LIN {X 0,Y 163.104,Z 333.396,A -85,B 0,C 180,E1 -26252.044,E2 -26252.044} C_VEL
LIN {X 0,Y 169.371,Z 321.967,A -85,B 0,C 180,E1 -26253.809,E2 -26253.809} C_VEL
LIN {X 0,Y 174.292,Z 311.209,A -85,B 0,C 180,E1 -26255.131,E2 -26255.131} C_VEL
LIN {X 0,Y 179.303,Z 297.656,A -85,B 0,C 180,E1 -26256.379,E2 -26256.379} C_VEL
LIN {X 0,Y 183.251,Z 283.24,A -85,B 0,C 180,E1 -26257.382,E2 -26257.382} C_VEL
LIN {X 0,Y 185.938,Z 269.575,A -85,B 0,C 180,E1 -26257.977,E2 -26257.977} C_VEL
LIN {X 0,Y 188.353,Z 247.435,A -85,B 0,C 180,E1 -26258.617,E2 -26258.617} C_VEL
LIN {X 0,Y 189.054,Z 239.838,A -85,B 0,C 180,E1 -26258.835,E2 -26258.835} C_VEL
LIN {X 0,Y 185.822,Z 232.857,A -85,B 0,C 180,E1 -26261.889,E2 -26261.889} C_VEL
LIN {X 0,Y 182.763,Z 226.917,A -85,B 0,C 180,E1 -26265.276,E2 -26265.276} C_VEL
LIN {X 0,Y 180.995,Z 223.675,A -85,B 0,C 180,E1 -26267.597,E2 -26267.597} C_VEL
LIN {X 0,Y 179.349,Z 220.559,A -85,B 0,C 180,E1 -26270.198,E2 -26270.198} C_VEL
LIN {X 0,Y 177.583,Z 217.018,A -85,B 0,C 180,E1 -26273.894,E2 -26273.894} C_VEL
LIN {X 0,Y 175.962,Z 213.489,A -85,B 0,C 180,E1 -26280.646,E2 -26280.646} C_VEL
LIN {X 0,Y 175.948,Z 212.764,A -85,B 0,C 180,E1 -26281.791,E2 -26281.791} C_VEL
LIN {X 0,Y 175.948,Z 213.169,A -85,B 0,C 180,E1 -26284.582,E2 -26284.582} C_VEL
LIN {X 0,Y 177.027,Z 216.627,A -85,B 0,C 180,E1 -26290.503,E2 -26290.503} C_VEL
LIN {X 0,Y 177.831,Z 217.67,A -85,B 0,C 180,E1 -26292.481,E2 -26292.481} C_VEL
LIN {X 0,Y 180.086,Z 221.968,A -85,B 0,C 180,E1 -26296.763,E2 -26296.763} C_VEL
LIN {X 0,Y 182.173,Z 225.802,A -85,B 0,C 180,E1 -26299.713,E2 -26299.713} C_VEL
LIN {X 0,Y 183.869,Z 229.479,A -85,B 0,C 180,E1 -26301.807,E2 -26301.807} C_VEL
LIN {X 0,Y 186.407,Z 236.279,A -85,B 0,C 180,E1 -26304.65,E2 -26304.65} C_VEL
LIN {X 0,Y 188.76,Z 243.058,A -85,B 0,C 180,E1 -26306.989,E2 -26306.989} C_VEL
LIN {X 0,Y 185.981,Z 270.935,A -85,B 0,C 180,E1 -26307.786,E2 -26307.786} C_VEL
LIN {X 0,Y 183.211,Z 285.581,A -85,B 0,C 180,E1 -26308.371,E2 -26308.371} C_VEL
LIN {X 0,Y 179.573,Z 298.889,A -85,B 0,C 180,E1 -26309.161,E2 -26309.161} C_VEL
LIN {X 0,Y 174.882,Z 311.931,A -85,B 0,C 180,E1 -26310.228,E2 -26310.228} C_VEL
LIN {X 0,Y 169.208,Z 324.559,A -85,B 0,C 180,E1 -26311.628,E2 -26311.628} C_VEL
LIN {X 0,Y 162.997,Z 336.072,A -85,B 0,C 180,E1 -26313.342,E2 -26313.342} C_VEL
LIN {X 0,Y 155.623,Z 347.616,A -85,B 0,C 180,E1 -26315.621,E2 -26315.621} C_VEL
LIN {X 0,Y 147.797,Z 358.182,A -85,B 0,C 180,E1 -26318.474,E2 -26318.474} C_VEL
LIN {X 0,Y 140.729,Z 366.499,A -85,B 0,C 180,E1 -26321.487,E2 -26321.487} C_VEL
LIN {X 0,Y 132.765,Z 374.701,A -85,B 0,C 180,E1 -26325.46,E2 -26325.46} C_VEL
LIN {X 0,Y 125.61,Z 381.317,A -85,B 0,C 180,E1 -26329.951,E2 -26329.951} C_VEL
LIN {X 0,Y 118.469,Z 387.209,A -85,B 0,C 180,E1 -26335.696,E2 -26335.696} C_VEL
LIN {X 0,Y 114.158,Z 390.634,A -85,B 0,C 180,E1 -26340.494,E2 -26340.494} C_VEL
LIN {X 0,Y 109.512,Z 393.899,A -85,B 0,C 180,E1 -26347.352,E2 -26347.352} C_VEL
LIN {X 0,Y 106.522,Z 395.797,A -85,B 0,C 180,E1 -26354.697,E2 -26354.697} C_VEL
LIN {X 0,Y 105.175,Z 396.381,A -85,B 0,C 180,E1 -26362.319,E2 -26362.319} C_VEL
LIN {X 0,Y 105.031,Z 396.178,A -85,B 0,C 180,E1 -26366.163,E2 -26366.163} C_VEL
LIN {X 0,Y 105.107,Z 395.641,A -85,B 0,C 180,E1 -26369.999,E2 -26369.999} C_VEL
LIN {X 0,Y 105.019,Z 394.753,A -85,B 0,C 180,E1 -26373.837,E2 -26373.837} C_VEL
LIN {X 0,Y 105.593,Z 391.925,A -85,B 0,C 180,E1 -26381.517,E2 -26381.517} C_VEL
LIN {X 0,Y 107.551,Z 387.625,A -85,B 0,C 180,E1 -26389.07,E2 -26389.07} C_VEL
LIN {X 0,Y 110.164,Z 383.371,A -85,B 0,C 180,E1 -26394.498,E2 -26394.498} C_VEL
LIN {X 0,Y 112.428,Z 379.759,A -85,B 0,C 180,E1 -26398.193,E2 -26398.193} C_VEL
LIN {X 0,Y 113.595,Z 377.02,A -85,B 0,C 180,E1 -26400.781,E2 -26400.781} C_VEL
LIN {X 0,Y 114.307,Z 372.208,A -85,B 0,C 180,E1 -26405.14,E2 -26405.14} C_VEL
LIN {X 0,Y 115.529,Z 366.929,A -85,B 0,C 180,E1 -26409.276,E2 -26409.276} C_VEL
LIN {X 0,Y 117.403,Z 363.367,A -85,B 0,C 180,E1 -26411.41,E2 -26411.41} C_VEL
LIN {X 0,Y 123.341,Z 354.399,A -85,B 0,C 180,E1 -26415.418,E2 -26415.418} C_VEL
LIN {X 0,Y 129.458,Z 344.175,A -85,B 0,C 180,E1 -26418.871,E2 -26418.871} C_VEL
LIN {X 0,Y 135.274,Z 332.907,A -85,B 0,C 180,E1 -26421.794,E2 -26421.794} C_VEL
LIN {X 0,Y 140.868,Z 320.442,A -85,B 0,C 180,E1 -26424.166,E2 -26424.166} C_VEL
LIN {X 0,Y 145.747,Z 307.43,A -85,B 0,C 180,E1 -26425.974,E2 -26425.974} C_VEL
LIN {X 0,Y 149.74,Z 293.962,A -85,B 0,C 180,E1 -26427.339,E2 -26427.339} C_VEL
LIN {X 0,Y 152.837,Z 279.632,A -85,B 0,C 180,E1 -26428.369,E2 -26428.369} C_VEL
LIN {X 0,Y 154.871,Z 265.326,A -85,B 0,C 180,E1 -26428.993,E2 -26428.993} C_VEL
LIN {X 0,Y 158.466,Z 223.489,A -85,B 0,C 180,E1 -26430.437,E2 -26430.437} C_VEL
LIN {X 0,Y 154.926,Z 212.982,A -85,B 0,C 180,E1 -26433.497,E2 -26433.497} C_VEL
LIN {X 0,Y 152.921,Z 208.654,A -85,B 0,C 180,E1 -26435.273,E2 -26435.273} C_VEL
LIN {X 0,Y 149.061,Z 201.739,A -85,B 0,C 180,E1 -26439.021,E2 -26439.021} C_VEL
LIN {X 0,Y 145.805,Z 196.184,A -85,B 0,C 180,E1 -26442.829,E2 -26442.829} C_VEL
LIN {X 0,Y 143.005,Z 191.844,A -85,B 0,C 180,E1 -26446.863,E2 -26446.863} C_VEL
LIN {X 0,Y 140.93,Z 188.345,A -85,B 0,C 180,E1 -26450.854,E2 -26450.854} C_VEL
LIN {X 0,Y 140.403,Z 187.555,A -85,B 0,C 180,E1 -26452.088,E2 -26452.088} C_VEL
LIN {X 0,Y 138.478,Z 184.233,A -85,B 0,C 180,E1 -26459.546,E2 -26459.546} C_VEL
LIN {X 0,Y 138.413,Z 182.933,A -85,B 0,C 180,E1 -26461.609,E2 -26461.609} C_VEL
LIN {X 0,Y 138.346,Z 183.294,A -85,B 0,C 180,E1 -26464.371,E2 -26464.371} C_VEL
LIN {X 0,Y 139.797,Z 187.241,A -85,B 0,C 180,E1 -26472.837,E2 -26472.837} C_VEL
LIN {X 0,Y 140.818,Z 188.256,A -85,B 0,C 180,E1 -26475.286,E2 -26475.286} C_VEL
LIN {X 0,Y 142.811,Z 191.691,A -85,B 0,C 180,E1 -26479.215,E2 -26479.215} C_VEL
LIN {X 0,Y 143.828,Z 193.178,A -85,B 0,C 180,E1 -26480.816,E2 -26480.816} C_VEL
LIN {X 0,Y 146.549,Z 197.585,A -85,B 0,C 180,E1 -26484.506,E2 -26484.506} C_VEL
LIN {X 0,Y 149.425,Z 202.393,A -85,B 0,C 180,E1 -26487.739,E2 -26487.739} C_VEL
LIN {X 0,Y 153.193,Z 209.339,A -85,B 0,C 180,E1 -26491.362,E2 -26491.362} C_VEL
LIN {X 0,Y 157.413,Z 217.975,A -85,B 0,C 180,E1 -26494.866,E2 -26494.866} C_VEL
LIN {X 0,Y 158.652,Z 220.72,A -85,B 0,C 180,E1 -26495.815,E2 -26495.815} C_VEL
LIN {X 0,Y 154.442,Z 267.31,A -85,B 0,C 180,E1 -26497.421,E2 -26497.421} C_VEL
LIN {X 0,Y 152.166,Z 281.337,A -85,B 0,C 180,E1 -26498.264,E2 -26498.264} C_VEL
LIN {X 0,Y 148.978,Z 294.723,A -85,B 0,C 180,E1 -26499.423,E2 -26499.423} C_VEL
LIN {X 0,Y 144.539,Z 308.698,A -85,B 0,C 180,E1 -26501.092,E2 -26501.092} C_VEL
LIN {X 0,Y 139.567,Z 321.183,A -85,B 0,C 180,E1 -26503.101,E2 -26503.101} C_VEL
LIN {X 0,Y 134.272,Z 332.561,A -85,B 0,C 180,E1 -26505.568,E2 -26505.568} C_VEL
LIN {X 0,Y 128.123,Z 343.987,A -85,B 0,C 180,E1 -26508.835,E2 -26508.835} C_VEL
LIN {X 0,Y 121.827,Z 354.21,A -85,B 0,C 180,E1 -26512.719,E2 -26512.719} C_VEL
LIN {X 0,Y 116.131,Z 362.66,A -85,B 0,C 180,E1 -26516.999,E2 -26516.999} C_VEL
LIN {X 0,Y 110.441,Z 370.728,A -85,B 0,C 180,E1 -26522.526,E2 -26522.526} C_VEL
LIN {X 0,Y 105.679,Z 377.239,A -85,B 0,C 180,E1 -26528.546,E2 -26528.546} C_VEL
LIN {X 0,Y 102.369,Z 381.755,A -85,B 0,C 180,E1 -26534.062,E2 -26534.062} C_VEL
LIN {X 0,Y 99.52,Z 386.369,A -85,B 0,C 180,E1 -26541.881,E2 -26541.881} C_VEL
LIN {X 0,Y 98.141,Z 389.507,A -85,B 0,C 180,E1 -26550.001,E2 -26550.001} C_VEL
LIN {X 0,Y 97.843,Z 390.569,A -85,B 0,C 180,E1 -26554.12,E2 -26554.12} C_VEL
LIN {X 0,Y 98.05,Z 391.703,A -85,B 0,C 180,E1 -26562.418,E2 -26562.418} C_VEL
LIN {X 0,Y 99.812,Z 391.512,A -85,B 0,C 180,E1 -26570.614,E2 -26570.614} C_VEL
LIN {X 0,Y 103.186,Z 389.978,A -85,B 0,C 180,E1 -26578.475,E2 -26578.475} C_VEL
LIN {X 0,Y 108.115,Z 387.062,A -85,B 0,C 180,E1 -26585.807,E2 -26585.807} C_VEL
LIN {X 0,Y 114.599,Z 382.674,A -85,B 0,C 180,E1 -26592.424,E2 -26592.424} C_VEL
LIN {X 0,Y 120.346,Z 378.294,A -85,B 0,C 180,E1 -26596.885,E2 -26596.885} C_VEL
LIN {X 0,Y 127.866,Z 371.916,A -85,B 0,C 180,E1 -26601.558,E2 -26601.558} C_VEL
LIN {X 0,Y 134.906,Z 365.106,A -85,B 0,C 180,E1 -26605.229,E2 -26605.229} C_VEL
LIN {X 0,Y 142.286,Z 357.096,A -85,B 0,C 180,E1 -26608.434,E2 -26608.434} C_VEL
LIN {X 0,Y 150.264,Z 347.31,A -85,B 0,C 180,E1 -26611.278,E2 -26611.278} C_VEL
LIN {X 0,Y 157.794,Z 336.411,A -85,B 0,C 180,E1 -26613.683,E2 -26613.683} C_VEL
LIN {X 0,Y 164.151,Z 325.597,A -85,B 0,C 180,E1 -26615.479,E2 -26615.479} C_VEL
LIN {X 0,Y 169.948,Z 313.913,A -85,B 0,C 180,E1 -26616.944,E2 -26616.944} C_VEL
LIN {X 0,Y 175.446,Z 300.22,A -85,B 0,C 180,E1 -26618.233,E2 -26618.233} C_VEL
LIN {X 0,Y 179.521,Z 286.575,A -85,B 0,C 180,E1 -26619.238,E2 -26619.238} C_VEL
LIN {X 0,Y 182.66,Z 272.102,A -85,B 0,C 180,E1 -26619.899,E2 -26619.899} C_VEL
LIN {X 0,Y 184.777,Z 255.073,A -85,B 0,C 180,E1 -26620.423,E2 -26620.423} C_VEL
LIN {X 0,Y 185.896,Z 243.533,A -85,B 0,C 180,E1 -26620.735,E2 -26620.735} C_VEL
LIN {X 0,Y 182.864,Z 236.776,A -85,B 0,C 180,E1 -26623.973,E2 -26623.973} C_VEL
LIN {X 0,Y 180.035,Z 231.055,A -85,B 0,C 180,E1 -26627.619,E2 -26627.619} C_VEL
LIN {X 0,Y 178.151,Z 227.388,A -85,B 0,C 180,E1 -26630.688,E2 -26630.688} C_VEL
LIN {X 0,Y 176.418,Z 223.824,A -85,B 0,C 180,E1 -26634.57,E2 -26634.57} C_VEL
LIN {X 0,Y 175.062,Z 220.259,A -85,B 0,C 180,E1 -26641.3,E2 -26641.3} C_VEL
LIN {X 0,Y 175.065,Z 219.76,A -85,B 0,C 180,E1 -26642.3,E2 -26642.3} C_VEL
LIN {X 0,Y 175.059,Z 220.213,A -85,B 0,C 180,E1 -26644.317,E2 -26644.317} C_VEL
LIN {X 0,Y 176.046,Z 223.603,A -85,B 0,C 180,E1 -26650.218,E2 -26650.218} C_VEL
LIN {X 0,Y 176.695,Z 224.506,A -85,B 0,C 180,E1 -26651.925,E2 -26651.925} C_VEL
LIN {X 0,Y 178.723,Z 228.592,A -85,B 0,C 180,E1 -26656.069,E2 -26656.069} C_VEL
LIN {X 0,Y 180.56,Z 232.171,A -85,B 0,C 180,E1 -26658.866,E2 -26658.866} C_VEL
LIN {X 0,Y 181.999,Z 235.567,A -85,B 0,C 180,E1 -26660.798,E2 -26660.798} C_VEL
LIN {X 0,Y 184.301,Z 242.191,A -85,B 0,C 180,E1 -26663.604,E2 -26663.604} C_VEL
LIN {X 0,Y 185.669,Z 246.321,A -85,B 0,C 180,E1 -26665.101,E2 -26665.101} C_VEL
LIN {X 0,Y 182.99,Z 271.487,A -85,B 0,C 180,E1 -26665.793,E2 -26665.793} C_VEL
LIN {X 0,Y 180.159,Z 285.904,A -85,B 0,C 180,E1 -26666.361,E2 -26666.361} C_VEL
LIN {X 0,Y 176.237,Z 299.649,A -85,B 0,C 180,E1 -26667.154,E2 -26667.154} C_VEL
LIN {X 0,Y 171.429,Z 312.489,A -85,B 0,C 180,E1 -26668.184,E2 -26668.184} C_VEL
LIN {X 0,Y 165.611,Z 324.977,A -85,B 0,C 180,E1 -26669.546,E2 -26669.546} C_VEL
LIN {X 0,Y 159.214,Z 336.387,A -85,B 0,C 180,E1 -26671.212,E2 -26671.212} C_VEL
LIN {X 0,Y 151.607,Z 347.848,A -85,B 0,C 180,E1 -26673.444,E2 -26673.444} C_VEL
LIN {X 0,Y 144.102,Z 357.592,A -85,B 0,C 180,E1 -26676.03,E2 -26676.03} C_VEL
LIN {X 0,Y 136.131,Z 366.605,A -85,B 0,C 180,E1 -26679.249,E2 -26679.249} C_VEL
LIN {X 0,Y 127.786,Z 374.742,A -85,B 0,C 180,E1 -26683.22,E2 -26683.22} C_VEL
LIN {X 0,Y 120.231,Z 381.317,A -85,B 0,C 180,E1 -26687.76,E2 -26687.76} C_VEL
LIN {X 0,Y 112.647,Z 387.172,A -85,B 0,C 180,E1 -26693.65,E2 -26693.65} C_VEL
LIN {X 0,Y 107.974,Z 390.572,A -85,B 0,C 180,E1 -26698.619,E2 -26698.619} C_VEL
LIN {X 0,Y 102.955,Z 393.793,A -85,B 0,C 180,E1 -26705.821,E2 -26705.821} C_VEL
LIN {X 0,Y 99.658,Z 395.658,A -85,B 0,C 180,E1 -26713.615,E2 -26713.615} C_VEL
LIN {X 0,Y 98.115,Z 396.209,A -85,B 0,C 180,E1 -26721.763,E2 -26721.763} C_VEL
LIN {X 0,Y 97.935,Z 395.991,A -85,B 0,C 180,E1 -26725.884,E2 -26725.884} C_VEL
LIN {X 0,Y 98.005,Z 395.438,A -85,B 0,C 180,E1 -26729.999,E2 -26729.999} C_VEL
LIN {X 0,Y 97.925,Z 394.533,A -85,B 0,C 180,E1 -26734.115,E2 -26734.115} C_VEL
LIN {X 0,Y 98.62,Z 391.671,A -85,B 0,C 180,E1 -26742.344,E2 -26742.344} C_VEL
LIN {X 0,Y 100.822,Z 387.334,A -85,B 0,C 180,E1 -26750.397,E2 -26750.397} C_VEL
LIN {X 0,Y 103.673,Z 383.041,A -85,B 0,C 180,E1 -26756.144,E2 -26756.144} C_VEL
LIN {X 0,Y 107.997,Z 376.757,A -85,B 0,C 180,E1 -26762.471,E2 -26762.471} C_VEL
LIN {X 0,Y 113.59,Z 368.924,A -85,B 0,C 180,E1 -26768.222,E2 -26768.222} C_VEL
LIN {X 0,Y 117.403,Z 363.367,A -85,B 0,C 180,E1 -26771.41,E2 -26771.41} C_VEL
LIN {X 0,Y 119.402,Z 359.663,A -85,B 0,C 180,E1 -26773.418,E2 -26773.418} C_VEL
LIN {X 0,Y 121.462,Z 353.381,A -85,B 0,C 180,E1 -26776.931,E2 -26776.931} C_VEL
LIN {X 0,Y 123.614,Z 346.643,A -85,B 0,C 180,E1 -26780.18,E2 -26780.18} C_VEL
LIN {X 0,Y 125.657,Z 342.225,A -85,B 0,C 180,E1 -26781.723,E2 -26781.723} C_VEL
LIN {X 0,Y 131.589,Z 330.916,A -85,B 0,C 180,E1 -26784.535,E2 -26784.535} C_VEL
LIN {X 0,Y 137.479,Z 318.039,A -85,B 0,C 180,E1 -26786.834,E2 -26786.834} C_VEL
LIN {X 0,Y 142.217,Z 305.453,A -85,B 0,C 180,E1 -26788.478,E2 -26788.478} C_VEL
LIN {X 0,Y 146.366,Z 291.429,A -85,B 0,C 180,E1 -26789.802,E2 -26789.802} C_VEL
LIN {X 0,Y 149.297,Z 277.579,A -85,B 0,C 180,E1 -26790.723,E2 -26790.723} C_VEL
LIN {X 0,Y 151.247,Z 263,A -85,B 0,C 180,E1 -26791.307,E2 -26791.307} C_VEL
LIN {X 0,Y 154.515,Z 225.964,A -85,B 0,C 180,E1 -26792.58,E2 -26792.58} C_VEL
LIN {X 0,Y 151.565,Z 216.879,A -85,B 0,C 180,E1 -26795.426,E2 -26795.426} C_VEL
LIN {X 0,Y 148.637,Z 210.986,A -85,B 0,C 180,E1 -26798.322,E2 -26798.322} C_VEL
LIN {X 0,Y 145.667,Z 205.538,A -85,B 0,C 180,E1 -26801.701,E2 -26801.701} C_VEL
LIN {X 0,Y 143.432,Z 201.744,A -85,B 0,C 180,E1 -26804.685,E2 -26804.685} C_VEL
LIN {X 0,Y 141.599,Z 198.533,A -85,B 0,C 180,E1 -26807.641,E2 -26807.641} C_VEL
LIN {X 0,Y 139.596,Z 194.873,A -85,B 0,C 180,E1 -26811.86,E2 -26811.86} C_VEL
LIN {X 0,Y 137.523,Z 190.884,A -85,B 0,C 180,E1 -26820.592,E2 -26820.592} C_VEL
LIN {X 0,Y 137.523,Z 189.96,A -85,B 0,C 180,E1 -26822.056,E2 -26822.056} C_VEL
LIN {X 0,Y 137.465,Z 190.509,A -85,B 0,C 180,E1 -26824.491,E2 -26824.491} C_VEL
LIN {X 0,Y 138.714,Z 194.154,A -85,B 0,C 180,E1 -26832.283,E2 -26832.283} C_VEL
LIN {X 0,Y 139.651,Z 195.224,A -85,B 0,C 180,E1 -26834.715,E2 -26834.715} C_VEL
LIN {X 0,Y 141.692,Z 198.729,A -85,B 0,C 180,E1 -26838.903,E2 -26838.903} C_VEL
LIN {X 0,Y 144.63,Z 203.761,A -85,B 0,C 180,E1 -26843.351,E2 -26843.351} C_VEL
LIN {X 0,Y 147.643,Z 209.116,A -85,B 0,C 180,E1 -26846.983,E2 -26846.983} C_VEL
LIN {X 0,Y 151.266,Z 216.339,A -85,B 0,C 180,E1 -26850.678,E2 -26850.678} C_VEL
LIN {X 0,Y 154.668,Z 223.78,A -85,B 0,C 180,E1 -26853.696,E2 -26853.696} C_VEL
LIN {X 0,Y 150.612,Z 267.23,A -85,B 0,C 180,E1 -26855.186,E2 -26855.186} C_VEL
LIN {X 0,Y 148.219,Z 281.466,A -85,B 0,C 180,E1 -26856.024,E2 -26856.024} C_VEL
LIN {X 0,Y 144.94,Z 294.764,A -85,B 0,C 180,E1 -26857.153,E2 -26857.153} C_VEL
LIN {X 0,Y 140.67,Z 307.884,A -85,B 0,C 180,E1 -26858.682,E2 -26858.682} C_VEL
LIN {X 0,Y 135.483,Z 320.559,A -85,B 0,C 180,E1 -26860.655,E2 -26860.655} C_VEL
LIN {X 0,Y 129.928,Z 332.078,A -85,B 0,C 180,E1 -26863.095,E2 -26863.095} C_VEL
LIN {X 0,Y 124.04,Z 342.643,A -85,B 0,C 180,E1 -26866.047,E2 -26866.047} C_VEL
LIN {X 0,Y 117.336,Z 353.131,A -85,B 0,C 180,E1 -26869.919,E2 -26869.919} C_VEL
LIN {X 0,Y 111.209,Z 361.787,A -85,B 0,C 180,E1 -26874.229,E2 -26874.229} C_VEL
LIN {X 0,Y 105.012,Z 370.089,A -85,B 0,C 180,E1 -26879.872,E2 -26879.872} C_VEL
LIN {X 0,Y 100.448,Z 375.875,A -85,B 0,C 180,E1 -26885.179,E2 -26885.179} C_VEL
LIN {X 0,Y 95.592,Z 382.074,A -85,B 0,C 180,E1 -26892.898,E2 -26892.898} C_VEL
LIN {X 0,Y 92.508,Z 386.632,A -85,B 0,C 180,E1 -26901.261,E2 -26901.261} C_VEL
LIN {X 0,Y 91.04,Z 389.732,A -85,B 0,C 180,E1 -26910.001,E2 -26910.001} C_VEL
LIN {X 0,Y 90.744,Z 390.777,A -85,B 0,C 180,E1 -26914.443,E2 -26914.443} C_VEL
LIN {X 0,Y 91.052,Z 391.877,A -85,B 0,C 180,E1 -26923.39,E2 -26923.39} C_VEL
LIN {X 0,Y 93.092,Z 391.65,A -85,B 0,C 180,E1 -26932.178,E2 -26932.178} C_VEL
LIN {X 0,Y 96.881,Z 390.08,A -85,B 0,C 180,E1 -26940.518,E2 -26940.518} C_VEL
LIN {X 0,Y 102.327,Z 387.127,A -85,B 0,C 180,E1 -26948.181,E2 -26948.181} C_VEL
LIN {X 0,Y 109.457,Z 382.637,A -85,B 0,C 180,E1 -26955.065,E2 -26955.065} C_VEL
LIN {X 0,Y 115.535,Z 378.277,A -85,B 0,C 180,E1 -26959.498,E2 -26959.498} C_VEL
LIN {X 0,Y 123.506,Z 371.855,A -85,B 0,C 180,E1 -26964.183,E2 -26964.183} C_VEL
LIN {X 0,Y 132.116,Z 363.844,A -85,B 0,C 180,E1 -26968.335,E2 -26968.335} C_VEL
LIN {X 0,Y 140.02,Z 355.434,A -85,B 0,C 180,E1 -26971.448,E2 -26971.448} C_VEL
LIN {X 0,Y 148.368,Z 345.281,A -85,B 0,C 180,E1 -26974.16,E2 -26974.16} C_VEL
LIN {X 0,Y 156.156,Z 333.853,A -85,B 0,C 180,E1 -26976.492,E2 -26976.492} C_VEL
LIN {X 0,Y 162.803,Z 322.461,A -85,B 0,C 180,E1 -26978.146,E2 -26978.146} C_VEL
LIN {X 0,Y 168.757,Z 309.962,A -85,B 0,C 180,E1 -26979.559,E2 -26979.559} C_VEL
LIN {X 0,Y 173.789,Z 296.759,A -85,B 0,C 180,E1 -26980.655,E2 -26980.655} C_VEL
LIN {X 0,Y 177.656,Z 283.154,A -85,B 0,C 180,E1 -26981.525,E2 -26981.525} C_VEL
LIN {X 0,Y 180.521,Z 268.984,A -85,B 0,C 180,E1 -26982.088,E2 -26982.088} C_VEL
LIN {X 0,Y 182.949,Z 247.322,A -85,B 0,C 180,E1 -26982.689,E2 -26982.689} C_VEL
LIN {X 0,Y 179.944,Z 240.491,A -85,B 0,C 180,E1 -26986.375,E2 -26986.375} C_VEL
LIN {X 0,Y 177.768,Z 236.075,A -85,B 0,C 180,E1 -26989.673,E2 -26989.673} C_VEL
LIN {X 0,Y 176.761,Z 233.861,A -85,B 0,C 180,E1 -26991.584,E2 -26991.584} C_VEL
LIN {X 0,Y 175.333,Z 230.66,A -85,B 0,C 180,E1 -26995.113,E2 -26995.113} C_VEL
LIN {X 0,Y 174.181,Z 227.13,A -85,B 0,C 180,E1 -27001.809,E2 -27001.809} C_VEL
LIN {X 0,Y 174.196,Z 226.822,A -85,B 0,C 180,E1 -27002.312,E2 -27002.312} C_VEL
LIN {X 0,Y 174.176,Z 227.232,A -85,B 0,C 180,E1 -27004.049,E2 -27004.049} C_VEL
LIN {X 0,Y 175.071,Z 230.567,A -85,B 0,C 180,E1 -27009.93,E2 -27009.93} C_VEL
LIN {X 0,Y 175.595,Z 231.377,A -85,B 0,C 180,E1 -27011.412,E2 -27011.412} C_VEL
LIN {X 0,Y 177.469,Z 235.394,A -85,B 0,C 180,E1 -27015.517,E2 -27015.517} C_VEL
LIN {X 0,Y 179.295,Z 239.222,A -85,B 0,C 180,E1 -27018.457,E2 -27018.457} C_VEL
LIN {X 0,Y 181.083,Z 244.267,A -85,B 0,C 180,E1 -27021,E2 -27021} C_VEL
LIN {X 0,Y 182.759,Z 249.639,A -85,B 0,C 180,E1 -27023.136,E2 -27023.136} C_VEL
LIN {X 0,Y 180.234,Z 272.031,A -85,B 0,C 180,E1 -27023.74,E2 -27023.74} C_VEL
LIN {X 0,Y 177.326,Z 286.234,A -85,B 0,C 180,E1 -27024.277,E2 -27024.277} C_VEL
LIN {X 0,Y 173.128,Z 300.412,A -85,B 0,C 180,E1 -27025.074,E2 -27025.074} C_VEL
LIN {X 0,Y 168.208,Z 313.05,A -85,B 0,C 180,E1 -27026.063,E2 -27026.063} C_VEL
LIN {X 0,Y 162.244,Z 325.398,A -85,B 0,C 180,E1 -27027.375,E2 -27027.375} C_VEL
LIN {X 0,Y 154.941,Z 337.871,A -85,B 0,C 180,E1 -27029.171,E2 -27029.171} C_VEL
LIN {X 0,Y 147.813,Z 348.086,A -85,B 0,C 180,E1 -27031.147,E2 -27031.147} C_VEL
LIN {X 0,Y 140.496,Z 357.217,A -85,B 0,C 180,E1 -27033.523,E2 -27033.523} C_VEL
LIN {X 0,Y 131.746,Z 366.703,A -85,B 0,C 180,E1 -27036.853,E2 -27036.853} C_VEL
LIN {X 0,Y 123.023,Z 374.784,A -85,B 0,C 180,E1 -27040.804,E2 -27040.804} C_VEL
LIN {X 0,Y 115.049,Z 381.318,A -85,B 0,C 180,E1 -27045.372,E2 -27045.372} C_VEL
LIN {X 0,Y 106.984,Z 387.134,A -85,B 0,C 180,E1 -27051.385,E2 -27051.385} C_VEL
LIN {X 0,Y 101.923,Z 390.504,A -85,B 0,C 180,E1 -27056.52,E2 -27056.52} C_VEL
LIN {X 0,Y 96.486,Z 393.686,A -85,B 0,C 180,E1 -27064.084,E2 -27064.084} C_VEL
LIN {X 0,Y 92.842,Z 395.519,A -85,B 0,C 180,E1 -27072.374,E2 -27072.374} C_VEL
LIN {X 0,Y 91.081,Z 396.038,A -85,B 0,C 180,E1 -27081.122,E2 -27081.122} C_VEL
LIN {X 0,Y 90.862,Z 395.804,A -85,B 0,C 180,E1 -27085.563,E2 -27085.563} C_VEL
LIN {X 0,Y 90.911,Z 395.234,A -85,B 0,C 180,E1 -27089.999,E2 -27089.999} C_VEL
LIN {X 0,Y 90.825,Z 394.312,A -85,B 0,C 180,E1 -27094.437,E2 -27094.437} C_VEL
LIN {X 0,Y 91.648,Z 391.415,A -85,B 0,C 180,E1 -27103.299,E2 -27103.299} C_VEL
LIN {X 0,Y 94.162,Z 387.044,A -85,B 0,C 180,E1 -27111.911,E2 -27111.911} C_VEL
LIN {X 0,Y 97.283,Z 382.711,A -85,B 0,C 180,E1 -27118.006,E2 -27118.006} C_VEL
LIN {X 0,Y 102.017,Z 376.386,A -85,B 0,C 180,E1 -27124.634,E2 -27124.634} C_VEL
LIN {X 0,Y 108.039,Z 368.506,A -85,B 0,C 180,E1 -27130.579,E2 -27130.579} C_VEL
LIN {X 0,Y 114.002,Z 360.267,A -85,B 0,C 180,E1 -27135.149,E2 -27135.149} C_VEL
LIN {X 0,Y 120.717,Z 350.342,A -85,B 0,C 180,E1 -27139.186,E2 -27139.186} C_VEL
LIN {X 0,Y 125.657,Z 342.225,A -85,B 0,C 180,E1 -27141.723,E2 -27141.723} C_VEL
LIN {X 0,Y 127.665,Z 337.74,A -85,B 0,C 180,E1 -27143.183,E2 -27143.183} C_VEL
LIN {X 0,Y 129.727,Z 330.204,A -85,B 0,C 180,E1 -27145.9,E2 -27145.9} C_VEL
LIN {X 0,Y 131.809,Z 322.362,A -85,B 0,C 180,E1 -27148.366,E2 -27148.366} C_VEL
LIN {X 0,Y 133.702,Z 317.246,A -85,B 0,C 180,E1 -27149.39,E2 -27149.39} C_VEL
LIN {X 0,Y 138.972,Z 303.467,A -85,B 0,C 180,E1 -27151.105,E2 -27151.105} C_VEL
LIN {X 0,Y 142.898,Z 290.17,A -85,B 0,C 180,E1 -27152.284,E2 -27152.284} C_VEL
LIN {X 0,Y 145.795,Z 276.687,A -85,B 0,C 180,E1 -27153.107,E2 -27153.107} C_VEL
LIN {X 0,Y 147.709,Z 262.134,A -85,B 0,C 180,E1 -27153.681,E2 -27153.681} C_VEL
LIN {X 0,Y 150.78,Z 228.515,A -85,B 0,C 180,E1 -27154.83,E2 -27154.83} C_VEL
LIN {X 0,Y 148.591,Z 221.499,A -85,B 0,C 180,E1 -27157.194,E2 -27157.194} C_VEL
LIN {X 0,Y 145.249,Z 214.542,A -85,B 0,C 180,E1 -27160.938,E2 -27160.938} C_VEL
LIN {X 0,Y 142.313,Z 208.97,A -85,B 0,C 180,E1 -27164.905,E2 -27164.905} C_VEL
LIN {X 0,Y 140.124,Z 205.101,A -85,B 0,C 180,E1 -27168.61,E2 -27168.61} C_VEL
LIN {X 0,Y 138.163,Z 201.308,A -85,B 0,C 180,E1 -27173.245,E2 -27173.245} C_VEL
LIN {X 0,Y 136.624,Z 197.937,A -85,B 0,C 180,E1 -27180.893,E2 -27180.893} C_VEL
LIN {X 0,Y 136.625,Z 197.058,A -85,B 0,C 180,E1 -27182.949,E2 -27182.949} C_VEL
LIN {X 0,Y 137.665,Z 201.086,A -85,B 0,C 180,E1 -27191.784,E2 -27191.784} C_VEL
LIN {X 0,Y 138.398,Z 201.907,A -85,B 0,C 180,E1 -27193.837,E2 -27193.837} C_VEL
LIN {X 0,Y 140.712,Z 206.199,A -85,B 0,C 180,E1 -27198.867,E2 -27198.867} C_VEL
LIN {X 0,Y 142.928,Z 210.285,A -85,B 0,C 180,E1 -27202.401,E2 -27202.401} C_VEL
LIN {X 0,Y 145.557,Z 215.239,A -85,B 0,C 180,E1 -27205.822,E2 -27205.822} C_VEL
LIN {X 0,Y 148.959,Z 222.456,A -85,B 0,C 180,E1 -27209.574,E2 -27209.574} C_VEL
LIN {X 0,Y 150.897,Z 226.881,A -85,B 0,C 180,E1 -27211.467,E2 -27211.467} C_VEL
LIN {X 0,Y 147.001,Z 267.257,A -85,B 0,C 180,E1 -27212.843,E2 -27212.843} C_VEL
LIN {X 0,Y 144.505,Z 281.586,A -85,B 0,C 180,E1 -27213.663,E2 -27213.663} C_VEL
LIN {X 0,Y 141.143,Z 294.79,A -85,B 0,C 180,E1 -27214.756,E2 -27214.756} C_VEL
LIN {X 0,Y 137.059,Z 307.061,A -85,B 0,C 180,E1 -27216.138,E2 -27216.138} C_VEL
LIN {X 0,Y 131.653,Z 319.93,A -85,B 0,C 180,E1 -27218.058,E2 -27218.058} C_VEL
LIN {X 0,Y 125.863,Z 331.587,A -85,B 0,C 180,E1 -27220.466,E2 -27220.466} C_VEL
LIN {X 0,Y 120.237,Z 341.3,A -85,B 0,C 180,E1 -27223.061,E2 -27223.061} C_VEL
LIN {X 0,Y 114.33,Z 350.415,A -85,B 0,C 180,E1 -27226.248,E2 -27226.248} C_VEL
LIN {X 0,Y 107.666,Z 359.555,A -85,B 0,C 180,E1 -27230.474,E2 -27230.474} C_VEL
LIN {X 0,Y 101.691,Z 367.173,A -85,B 0,C 180,E1 -27235.239,E2 -27235.239} C_VEL
LIN {X 0,Y 95.613,Z 374.441,A -85,B 0,C 180,E1 -27241.46,E2 -27241.46} C_VEL
LIN {X 0,Y 90.037,Z 380.977,A -85,B 0,C 180,E1 -27249.437,E2 -27249.437} C_VEL
LIN {X 0,Y 86.091,Z 386.041,A -85,B 0,C 180,E1 -27258.568,E2 -27258.568} C_VEL
LIN {X 0,Y 84.515,Z 388.598,A -85,B 0,C 180,E1 -27265.231,E2 -27265.231} C_VEL
LIN {X 0,Y 83.933,Z 389.958,A -85,B 0,C 180,E1 -27270.001,E2 -27270.001} C_VEL
LIN {X 0,Y 83.618,Z 390.986,A -85,B 0,C 180,E1 -27274.822,E2 -27274.822} C_VEL
LIN {X 0,Y 84.094,Z 392.051,A -85,B 0,C 180,E1 -27284.521,E2 -27284.521} C_VEL
LIN {X 0,Y 86.454,Z 391.788,A -85,B 0,C 180,E1 -27293.983,E2 -27293.983} C_VEL
LIN {X 0,Y 90.711,Z 390.183,A -85,B 0,C 180,E1 -27302.844,E2 -27302.844} C_VEL
LIN {X 0,Y 96.742,Z 387.192,A -85,B 0,C 180,E1 -27310.831,E2 -27310.831} C_VEL
LIN {X 0,Y 104.371,Z 382.726,A -85,B 0,C 180,E1 -27317.792,E2 -27317.792} C_VEL
LIN {X 0,Y 110.965,Z 378.262,A -85,B 0,C 180,E1 -27322.345,E2 -27322.345} C_VEL
LIN {X 0,Y 119.414,Z 371.795,A -85,B 0,C 180,E1 -27327.001,E2 -27327.001} C_VEL
LIN {X 0,Y 127.286,Z 364.832,A -85,B 0,C 180,E1 -27330.599,E2 -27330.599} C_VEL
LIN {X 0,Y 135.311,Z 356.763,A -85,B 0,C 180,E1 -27333.633,E2 -27333.633} C_VEL
LIN {X 0,Y 143.921,Z 346.846,A -85,B 0,C 180,E1 -27336.293,E2 -27336.293} C_VEL
LIN {X 0,Y 151.927,Z 335.782,A -85,B 0,C 180,E1 -27338.586,E2 -27338.586} C_VEL
LIN {X 0,Y 158.736,Z 324.776,A -85,B 0,C 180,E1 -27340.193,E2 -27340.193} C_VEL
LIN {X 0,Y 164.845,Z 312.83,A -85,B 0,C 180,E1 -27341.552,E2 -27341.552} C_VEL
LIN {X 0,Y 170.116,Z 300.106,A -85,B 0,C 180,E1 -27342.622,E2 -27342.622} C_VEL
LIN {X 0,Y 174.467,Z 286.063,A -85,B 0,C 180,E1 -27343.555,E2 -27343.555} C_VEL
LIN {X 0,Y 177.631,Z 271.949,A -85,B 0,C 180,E1 -27344.12,E2 -27344.12} C_VEL
LIN {X 0,Y 179.936,Z 253.876,A -85,B 0,C 180,E1 -27344.635,E2 -27344.635} C_VEL
LIN {X 0,Y 180.201,Z 251.376,A -85,B 0,C 180,E1 -27344.692,E2 -27344.692} C_VEL
LIN {X 0,Y 177.819,Z 245.788,A -85,B 0,C 180,E1 -27348.024,E2 -27348.024} C_VEL
LIN {X 0,Y 175.737,Z 240.938,A -85,B 0,C 180,E1 -27351.809,E2 -27351.809} C_VEL
LIN {X 0,Y 174.36,Z 237.635,A -85,B 0,C 180,E1 -27355.376,E2 -27355.376} C_VEL
LIN {X 0,Y 173.303,Z 234.155,A -85,B 0,C 180,E1 -27362.071,E2 -27362.071} C_VEL
LIN {X 0,Y 173.306,Z 234.099,A -85,B 0,C 180,E1 -27363.523,E2 -27363.523} C_VEL
LIN {X 0,Y 174.1,Z 237.526,A -85,B 0,C 180,E1 -27369.639,E2 -27369.639} C_VEL
LIN {X 0,Y 174.569,Z 238.44,A -85,B 0,C 180,E1 -27371.084,E2 -27371.084} C_VEL
LIN {X 0,Y 176.187,Z 242.124,A -85,B 0,C 180,E1 -27374.874,E2 -27374.874} C_VEL
LIN {X 0,Y 177.856,Z 245.844,A -85,B 0,C 180,E1 -27377.758,E2 -27377.758} C_VEL
LIN {X 0,Y 179.59,Z 251.535,A -85,B 0,C 180,E1 -27380.457,E2 -27380.457} C_VEL
LIN {X 0,Y 180.032,Z 253.142,A -85,B 0,C 180,E1 -27381.094,E2 -27381.094} C_VEL
LIN {X 0,Y 177.858,Z 271.696,A -85,B 0,C 180,E1 -27381.59,E2 -27381.59} C_VEL
LIN {X 0,Y 174.76,Z 286.481,A -85,B 0,C 180,E1 -27382.129,E2 -27382.129} C_VEL
LIN {X 0,Y 170.65,Z 300.05,A -85,B 0,C 180,E1 -27382.855,E2 -27382.855} C_VEL
LIN {X 0,Y 165.228,Z 313.61,A -85,B 0,C 180,E1 -27383.864,E2 -27383.864} C_VEL
LIN {X 0,Y 159.117,Z 325.82,A -85,B 0,C 180,E1 -27385.114,E2 -27385.114} C_VEL
LIN {X 0,Y 151.615,Z 338.164,A -85,B 0,C 180,E1 -27386.833,E2 -27386.833} C_VEL
LIN {X 0,Y 144.273,Z 348.31,A -85,B 0,C 180,E1 -27388.736,E2 -27388.736} C_VEL
LIN {X 0,Y 136.23,Z 357.92,A -85,B 0,C 180,E1 -27391.197,E2 -27391.197} C_VEL
LIN {X 0,Y 127.604,Z 366.794,A -85,B 0,C 180,E1 -27394.294,E2 -27394.294} C_VEL
LIN {X 0,Y 118.5,Z 374.828,A -85,B 0,C 180,E1 -27398.202,E2 -27398.202} C_VEL
LIN {X 0,Y 110.096,Z 381.32,A -85,B 0,C 180,E1 -27402.767,E2 -27402.767} C_VEL
LIN {X 0,Y 101.501,Z 387.098,A -85,B 0,C 180,E1 -27408.868,E2 -27408.868} C_VEL
LIN {X 0,Y 96.034,Z 390.432,A -85,B 0,C 180,E1 -27414.164,E2 -27414.164} C_VEL
LIN {X 0,Y 90.122,Z 393.579,A -85,B 0,C 180,E1 -27422.101,E2 -27422.101} C_VEL
LIN {X 0,Y 86.063,Z 395.379,A -85,B 0,C 180,E1 -27430.934,E2 -27430.934} C_VEL
LIN {X 0,Y 84.047,Z 395.866,A -85,B 0,C 180,E1 -27440.372,E2 -27440.372} C_VEL
LIN {X 0,Y 83.776,Z 395.616,A -85,B 0,C 180,E1 -27445.187,E2 -27445.187} C_VEL
LIN {X 0,Y 83.809,Z 395.031,A -85,B 0,C 180,E1 -27449.999,E2 -27449.999} C_VEL
LIN {X 0,Y 83.748,Z 394.093,A -85,B 0,C 180,E1 -27454.813,E2 -27454.813} C_VEL
LIN {X 0,Y 84.718,Z 391.161,A -85,B 0,C 180,E1 -27464.41,E2 -27464.41} C_VEL
LIN {X 0,Y 87.584,Z 386.754,A -85,B 0,C 180,E1 -27473.653,E2 -27473.653} C_VEL
LIN {X 0,Y 92.398,Z 380.745,A -85,B 0,C 180,E1 -27482.169,E2 -27482.169} C_VEL
LIN {X 0,Y 97.964,Z 373.958,A -85,B 0,C 180,E1 -27488.882,E2 -27488.882} C_VEL
LIN {X 0,Y 104.75,Z 365.503,A -85,B 0,C 180,E1 -27494.786,E2 -27494.786} C_VEL
LIN {X 0,Y 111.396,Z 356.689,A -85,B 0,C 180,E1 -27499.207,E2 -27499.207} C_VEL
LIN {X 0,Y 118.641,Z 346,A -85,B 0,C 180,E1 -27503.101,E2 -27503.101} C_VEL
LIN {X 0,Y 125.084,Z 334.931,A -85,B 0,C 180,E1 -27506.122,E2 -27506.122} C_VEL
LIN {X 0,Y 130.961,Z 323.368,A -85,B 0,C 180,E1 -27508.421,E2 -27508.421} C_VEL
LIN {X 0,Y 133.702,Z 317.246,A -85,B 0,C 180,E1 -27509.39,E2 -27509.39} C_VEL
LIN {X 0,Y 135.504,Z 312.074,A -85,B 0,C 180,E1 -27510.342,E2 -27510.342} C_VEL
LIN {X 0,Y 137.153,Z 303.541,A -85,B 0,C 180,E1 -27512.363,E2 -27512.363} C_VEL
LIN {X 0,Y 138.454,Z 294.75,A -85,B 0,C 180,E1 -27514.197,E2 -27514.197} C_VEL
LIN {X 0,Y 139.623,Z 289.176,A -85,B 0,C 180,E1 -27514.847,E2 -27514.847} C_VEL
LIN {X 0,Y 142.541,Z 275.601,A -85,B 0,C 180,E1 -27515.633,E2 -27515.633} C_VEL
LIN {X 0,Y 144.594,Z 259.778,A -85,B 0,C 180,E1 -27516.204,E2 -27516.204} C_VEL
LIN {X 0,Y 147.28,Z 231.146,A -85,B 0,C 180,E1 -27517.188,E2 -27517.188} C_VEL
LIN {X 0,Y 145.818,Z 226.34,A -85,B 0,C 180,E1 -27518.96,E2 -27518.96} C_VEL
LIN {X 0,Y 142.816,Z 219.803,A -85,B 0,C 180,E1 -27522.712,E2 -27522.712} C_VEL
LIN {X 0,Y 140.196,Z 214.627,A -85,B 0,C 180,E1 -27526.71,E2 -27526.71} C_VEL
LIN {X 0,Y 138.668,Z 211.631,A -85,B 0,C 180,E1 -27529.644,E2 -27529.644} C_VEL
LIN {X 0,Y 136.972,Z 208.076,A -85,B 0,C 180,E1 -27534.11,E2 -27534.11} C_VEL
LIN {X 0,Y 135.727,Z 204.749,A -85,B 0,C 180,E1 -27541.641,E2 -27541.641} C_VEL
LIN {X 0,Y 135.751,Z 204.164,A -85,B 0,C 180,E1 -27542.968,E2 -27542.968} C_VEL
LIN {X 0,Y 136.674,Z 208.04,A -85,B 0,C 180,E1 -27551.426,E2 -27551.426} C_VEL
LIN {X 0,Y 137.296,Z 208.897,A -85,B 0,C 180,E1 -27553.32,E2 -27553.32} C_VEL
LIN {X 0,Y 139.386,Z 213.078,A -85,B 0,C 180,E1 -27558.196,E2 -27558.196} C_VEL
LIN {X 0,Y 141.358,Z 216.972,A -85,B 0,C 180,E1 -27561.569,E2 -27561.569} C_VEL
LIN {X 0,Y 143.901,Z 222.167,A -85,B 0,C 180,E1 -27565.107,E2 -27565.107} C_VEL
LIN {X 0,Y 146.844,Z 228.998,A -85,B 0,C 180,E1 -27568.595,E2 -27568.595} C_VEL
LIN {X 0,Y 147.36,Z 230.246,A -85,B 0,C 180,E1 -27569.153,E2 -27569.153} C_VEL
LIN {X 0,Y 143.524,Z 267.926,A -85,B 0,C 180,E1 -27570.396,E2 -27570.396} C_VEL
LIN {X 0,Y 140.881,Z 282.403,A -85,B 0,C 180,E1 -27571.227,E2 -27571.227} C_VEL
LIN {X 0,Y 137.253,Z 295.939,A -85,B 0,C 180,E1 -27572.343,E2 -27572.343} C_VEL
LIN {X 0,Y 132.32,Z 309.754,A -85,B 0,C 180,E1 -27573.913,E2 -27573.913} C_VEL
LIN {X 0,Y 126.731,Z 322.135,A -85,B 0,C 180,E1 -27575.803,E2 -27575.803} C_VEL
LIN {X 0,Y 120.719,Z 333.433,A -85,B 0,C 180,E1 -27578.193,E2 -27578.193} C_VEL
LIN {X 0,Y 114.307,Z 343.823,A -85,B 0,C 180,E1 -27581.135,E2 -27581.135} C_VEL
LIN {X 0,Y 106.912,Z 354.171,A -85,B 0,C 180,E1 -27585.037,E2 -27585.037} C_VEL
LIN {X 0,Y 100.079,Z 362.708,A -85,B 0,C 180,E1 -27589.491,E2 -27589.491} C_VEL
LIN {X 0,Y 93.044,Z 370.883,A -85,B 0,C 180,E1 -27595.494,E2 -27595.494} C_VEL
LIN {X 0,Y 87.788,Z 376.6,A -85,B 0,C 180,E1 -27601.294,E2 -27601.294} C_VEL
LIN {X 0,Y 83.45,Z 381.296,A -85,B 0,C 180,E1 -27607.73,E2 -27607.73} C_VEL
LIN {X 0,Y 79.281,Z 386.168,A -85,B 0,C 180,E1 -27617.197,E2 -27617.197} C_VEL
LIN {X 0,Y 77.443,Z 388.841,A -85,B 0,C 180,E1 -27624.794,E2 -27624.794} C_VEL
LIN {X 0,Y 76.809,Z 390.184,A -85,B 0,C 180,E1 -27630.001,E2 -27630.001} C_VEL
LIN {X 0,Y 76.512,Z 391.194,A -85,B 0,C 180,E1 -27635.271,E2 -27635.271} C_VEL
LIN {X 0,Y 77.164,Z 392.224,A -85,B 0,C 180,E1 -27645.858,E2 -27645.858} C_VEL
LIN {X 0,Y 79.913,Z 391.927,A -85,B 0,C 180,E1 -27656.088,E2 -27656.088} C_VEL
LIN {X 0,Y 84.727,Z 390.286,A -85,B 0,C 180,E1 -27665.496,E2 -27665.496} C_VEL
LIN {X 0,Y 91.396,Z 387.258,A -85,B 0,C 180,E1 -27673.795,E2 -27673.795} C_VEL
LIN {X 0,Y 99.661,Z 382.748,A -85,B 0,C 180,E1 -27680.87,E2 -27680.87} C_VEL
LIN {X 0,Y 106.701,Z 378.247,A -85,B 0,C 180,E1 -27685.42,E2 -27685.42} C_VEL
LIN {X 0,Y 115.621,Z 371.734,A -85,B 0,C 180,E1 -27690.019,E2 -27690.019} C_VEL
LIN {X 0,Y 125.115,Z 363.623,A -85,B 0,C 180,E1 -27693.996,E2 -27693.996} C_VEL
LIN {X 0,Y 133.738,Z 355.1,A -85,B 0,C 180,E1 -27696.874,E2 -27696.874} C_VEL
LIN {X 0,Y 142.679,Z 344.759,A -85,B 0,C 180,E1 -27699.374,E2 -27699.374} C_VEL
LIN {X 0,Y 150.225,Z 334.319,A -85,B 0,C 180,E1 -27701.328,E2 -27701.328} C_VEL
LIN {X 0,Y 157.236,Z 322.957,A -85,B 0,C 180,E1 -27702.824,E2 -27702.824} C_VEL
LIN {X 0,Y 163.51,Z 310.503,A -85,B 0,C 180,E1 -27704.097,E2 -27704.097} C_VEL
LIN {X 0,Y 168.601,Z 297.877,A -85,B 0,C 180,E1 -27705.057,E2 -27705.057} C_VEL
LIN {X 0,Y 172.781,Z 284.087,A -85,B 0,C 180,E1 -27705.874,E2 -27705.874} C_VEL
LIN {X 0,Y 175.793,Z 270.096,A -85,B 0,C 180,E1 -27706.381,E2 -27706.381} C_VEL
LIN {X 0,Y 177.655,Z 255.483,A -85,B 0,C 180,E1 -27706.778,E2 -27706.778} C_VEL
LIN {X 0,Y 175.59,Z 250.353,A -85,B 0,C 180,E1 -27710.206,E2 -27710.206} C_VEL
LIN {X 0,Y 174.256,Z 247.171,A -85,B 0,C 180,E1 -27713.05,E2 -27713.05} C_VEL
LIN {X 0,Y 173.205,Z 244.389,A -85,B 0,C 180,E1 -27716.219,E2 -27716.219} C_VEL
LIN {X 0,Y 172.428,Z 241.195,A -85,B 0,C 180,E1 -27722.336,E2 -27722.336} C_VEL
LIN {X 0,Y 172.43,Z 241.174,A -85,B 0,C 180,E1 -27723.34,E2 -27723.34} C_VEL
LIN {X 0,Y 173.134,Z 244.49,A -85,B 0,C 180,E1 -27729.344,E2 -27729.344} C_VEL
LIN {X 0,Y 173.519,Z 245.384,A -85,B 0,C 180,E1 -27730.645,E2 -27730.645} C_VEL
LIN {X 0,Y 174.982,Z 248.909,A -85,B 0,C 180,E1 -27734.32,E2 -27734.32} C_VEL
LIN {X 0,Y 176.396,Z 252.431,A -85,B 0,C 180,E1 -27736.981,E2 -27736.981} C_VEL
LIN {X 0,Y 177.562,Z 256.734,A -85,B 0,C 180,E1 -27739.026,E2 -27739.026} C_VEL
LIN {X 0,Y 175.376,Z 273.512,A -85,B 0,C 180,E1 -27739.459,E2 -27739.459} C_VEL
LIN {X 0,Y 172.123,Z 287.971,A -85,B 0,C 180,E1 -27739.972,E2 -27739.972} C_VEL
LIN {X 0,Y 167.635,Z 301.939,A -85,B 0,C 180,E1 -27740.7,E2 -27740.7} C_VEL
LIN {X 0,Y 162.501,Z 314.171,A -85,B 0,C 180,E1 -27741.588,E2 -27741.588} C_VEL
LIN {X 0,Y 156.249,Z 326.241,A -85,B 0,C 180,E1 -27742.767,E2 -27742.767} C_VEL
LIN {X 0,Y 148.551,Z 338.441,A -85,B 0,C 180,E1 -27744.394,E2 -27744.394} C_VEL
LIN {X 0,Y 141.001,Z 348.518,A -85,B 0,C 180,E1 -27746.209,E2 -27746.209} C_VEL
LIN {X 0,Y 132.195,Z 358.574,A -85,B 0,C 180,E1 -27748.726,E2 -27748.726} C_VEL
LIN {X 0,Y 123.735,Z 366.884,A -85,B 0,C 180,E1 -27751.571,E2 -27751.571} C_VEL
LIN {X 0,Y 114.235,Z 374.872,A -85,B 0,C 180,E1 -27755.395,E2 -27755.395} C_VEL
LIN {X 0,Y 105.397,Z 381.323,A -85,B 0,C 180,E1 -27759.929,E2 -27759.929} C_VEL
LIN {X 0,Y 96.256,Z 387.062,A -85,B 0,C 180,E1 -27766.081,E2 -27766.081} C_VEL
LIN {X 0,Y 90.316,Z 390.36,A -85,B 0,C 180,E1 -27771.499,E2 -27771.499} C_VEL
LIN {X 0,Y 83.886,Z 393.474,A -85,B 0,C 180,E1 -27779.821,E2 -27779.821} C_VEL
LIN {X 0,Y 79.334,Z 395.24,A -85,B 0,C 180,E1 -27789.245,E2 -27789.245} C_VEL
LIN {X 0,Y 77.042,Z 395.694,A -85,B 0,C 180,E1 -27799.487,E2 -27799.487} C_VEL
LIN {X 0,Y 76.693,Z 395.428,A -85,B 0,C 180,E1 -27804.741,E2 -27804.741} C_VEL
LIN {X 0,Y 76.729,Z 394.828,A -85,B 0,C 180,E1 -27809.999,E2 -27809.999} C_VEL
LIN {X 0,Y 76.65,Z 393.872,A -85,B 0,C 180,E1 -27815.26,E2 -27815.26} C_VEL
LIN {X 0,Y 77.835,Z 390.906,A -85,B 0,C 180,E1 -27825.716,E2 -27825.716} C_VEL
LIN {X 0,Y 81.099,Z 386.463,A -85,B 0,C 180,E1 -27835.676,E2 -27835.676} C_VEL
LIN {X 0,Y 84.902,Z 382.051,A -85,B 0,C 180,E1 -27842.55,E2 -27842.55} C_VEL
LIN {X 0,Y 90.613,Z 375.644,A -85,B 0,C 180,E1 -27849.781,E2 -27849.781} C_VEL
LIN {X 0,Y 97.612,Z 367.671,A -85,B 0,C 180,E1 -27856.053,E2 -27856.053} C_VEL
LIN {X 0,Y 104.407,Z 359.327,A -85,B 0,C 180,E1 -27860.723,E2 -27860.723} C_VEL
LIN {X 0,Y 111.874,Z 349.277,A -85,B 0,C 180,E1 -27864.752,E2 -27864.752} C_VEL
LIN {X 0,Y 118.134,Z 339.616,A -85,B 0,C 180,E1 -27867.628,E2 -27867.628} C_VEL
LIN {X 0,Y 124.519,Z 328.216,A -85,B 0,C 180,E1 -27870.201,E2 -27870.201} C_VEL
LIN {X 0,Y 130.213,Z 316.403,A -85,B 0,C 180,E1 -27872.104,E2 -27872.104} C_VEL
LIN {X 0,Y 135.306,Z 303.483,A -85,B 0,C 180,E1 -27873.634,E2 -27873.634} C_VEL
LIN {X 0,Y 139.353,Z 290.252,A -85,B 0,C 180,E1 -27874.774,E2 -27874.774} C_VEL
LIN {X 0,Y 139.623,Z 289.176,A -85,B 0,C 180,E1 -27874.847,E2 -27874.847} C_VEL
LIN {X 0,Y 140.692,Z 283.535,A -85,B 0,C 180,E1 -27875.439,E2 -27875.439} C_VEL
LIN {X 0,Y 141.178,Z 274.341,A -85,B 0,C 180,E1 -27876.935,E2 -27876.935} C_VEL
LIN {X 0,Y 141.256,Z 265.042,A -85,B 0,C 180,E1 -27878.345,E2 -27878.345} C_VEL
LIN {X 0,Y 141.589,Z 259.235,A -85,B 0,C 180,E1 -27878.778,E2 -27878.778} C_VEL
LIN {X 0,Y 144.066,Z 234.059,A -85,B 0,C 180,E1 -27879.6,E2 -27879.6} C_VEL
LIN {X 0,Y 143.286,Z 231.422,A -85,B 0,C 180,E1 -27880.666,E2 -27880.666} C_VEL
LIN {X 0,Y 140.436,Z 224.771,A -85,B 0,C 180,E1 -27884.699,E2 -27884.699} C_VEL
LIN {X 0,Y 138.286,Z 220.327,A -85,B 0,C 180,E1 -27888.457,E2 -27888.457} C_VEL
LIN {X 0,Y 137.26,Z 218.144,A -85,B 0,C 180,E1 -27890.7,E2 -27890.7} C_VEL
LIN {X 0,Y 135.946,Z 215.011,A -85,B 0,C 180,E1 -27894.55,E2 -27894.55} C_VEL
LIN {X 0,Y 134.843,Z 211.736,A -85,B 0,C 180,E1 -27902.097,E2 -27902.097} C_VEL
LIN {X 0,Y 134.867,Z 211.352,A -85,B 0,C 180,E1 -27902.988,E2 -27902.988} C_VEL
LIN {X 0,Y 135.724,Z 215.058,A -85,B 0,C 180,E1 -27911.197,E2 -27911.197} C_VEL
LIN {X 0,Y 136.15,Z 215.702,A -85,B 0,C 180,E1 -27912.596,E2 -27912.596} C_VEL
LIN {X 0,Y 138.061,Z 219.854,A -85,B 0,C 180,E1 -27917.461,E2 -27917.461} C_VEL
LIN {X 0,Y 140.118,Z 224.212,A -85,B 0,C 180,E1 -27921.193,E2 -27921.193} C_VEL
LIN {X 0,Y 142.661,Z 230.086,A -85,B 0,C 180,E1 -27924.915,E2 -27924.915} C_VEL
LIN {X 0,Y 144.056,Z 233.601,A -85,B 0,C 180,E1 -27926.71,E2 -27926.71} C_VEL
LIN {X 0,Y 140.563,Z 267.31,A -85,B 0,C 180,E1 -27927.811,E2 -27927.811} C_VEL
LIN {X 0,Y 137.856,Z 281.881,A -85,B 0,C 180,E1 -27928.583,E2 -27928.583} C_VEL
LIN {X 0,Y 134.351,Z 294.843,A -85,B 0,C 180,E1 -27929.582,E2 -27929.582} C_VEL
LIN {X 0,Y 129.98,Z 307.173,A -85,B 0,C 180,E1 -27930.868,E2 -27930.868} C_VEL
LIN {X 0,Y 124.901,Z 318.663,A -85,B 0,C 180,E1 -27932.433,E2 -27932.433} C_VEL
LIN {X 0,Y 119.269,Z 329.422,A -85,B 0,C 180,E1 -27934.417,E2 -27934.417} C_VEL
LIN {X 0,Y 112.394,Z 340.54,A -85,B 0,C 180,E1 -27937.132,E2 -27937.132} C_VEL
LIN {X 0,Y 104.565,Z 351.454,A -85,B 0,C 180,E1 -27940.877,E2 -27940.877} C_VEL
LIN {X 0,Y 97.158,Z 360.475,A -85,B 0,C 180,E1 -27945.149,E2 -27945.149} C_VEL
LIN {X 0,Y 90.427,Z 367.987,A -85,B 0,C 180,E1 -27950.12,E2 -27950.12} C_VEL
LIN {X 0,Y 83.455,Z 375.162,A -85,B 0,C 180,E1 -27956.813,E2 -27956.813} C_VEL
LIN {X 0,Y 76.937,Z 381.615,A -85,B 0,C 180,E1 -27965.729,E2 -27965.729} C_VEL
LIN {X 0,Y 72.39,Z 386.448,A -85,B 0,C 180,E1 -27975.954,E2 -27975.954} C_VEL
LIN {X 0,Y 70.388,Z 389.084,A -85,B 0,C 180,E1 -27984.271,E2 -27984.271} C_VEL
LIN {X 0,Y 69.708,Z 390.408,A -85,B 0,C 180,E1 -27990.001,E2 -27990.001} C_VEL
LIN {X 0,Y 69.405,Z 391.402,A -85,B 0,C 180,E1 -27995.813,E2 -27995.813} C_VEL
LIN {X 0,Y 70.266,Z 392.398,A -85,B 0,C 180,E1 -28007.462,E2 -28007.462} C_VEL
LIN {X 0,Y 73.506,Z 392.065,A -85,B 0,C 180,E1 -28018.559,E2 -28018.559} C_VEL
LIN {X 0,Y 78.959,Z 390.389,A -85,B 0,C 180,E1 -28028.541,E2 -28028.541} C_VEL
LIN {X 0,Y 86.324,Z 387.324,A -85,B 0,C 180,E1 -28037.116,E2 -28037.116} C_VEL
LIN {X 0,Y 95.255,Z 382.762,A -85,B 0,C 180,E1 -28044.253,E2 -28044.253} C_VEL
LIN {X 0,Y 102.779,Z 378.232,A -85,B 0,C 180,E1 -28048.733,E2 -28048.733} C_VEL
LIN {X 0,Y 112.173,Z 371.674,A -85,B 0,C 180,E1 -28053.229,E2 -28053.229} C_VEL
LIN {X 0,Y 122.122,Z 363.504,A -85,B 0,C 180,E1 -28057.043,E2 -28057.043} C_VEL
LIN {X 0,Y 131.077,Z 354.922,A -85,B 0,C 180,E1 -28059.77,E2 -28059.77} C_VEL
LIN {X 0,Y 140.297,Z 344.492,A -85,B 0,C 180,E1 -28062.136,E2 -28062.136} C_VEL
LIN {X 0,Y 148.085,Z 333.969,A -85,B 0,C 180,E1 -28063.956,E2 -28063.956} C_VEL
LIN {X 0,Y 155.279,Z 322.501,A -85,B 0,C 180,E1 -28065.341,E2 -28065.341} C_VEL
LIN {X 0,Y 161.695,Z 309.898,A -85,B 0,C 180,E1 -28066.537,E2 -28066.537} C_VEL
LIN {X 0,Y 167.261,Z 296.008,A -85,B 0,C 180,E1 -28067.509,E2 -28067.509} C_VEL
LIN {X 0,Y 171.065,Z 283.351,A -85,B 0,C 180,E1 -28068.174,E2 -28068.174} C_VEL
LIN {X 0,Y 174.014,Z 269.573,A -85,B 0,C 180,E1 -28068.635,E2 -28068.635} C_VEL
LIN {X 0,Y 175.321,Z 259.786,A -85,B 0,C 180,E1 -28068.935,E2 -28068.935} C_VEL
LIN {X 0,Y 173.529,Z 255.025,A -85,B 0,C 180,E1 -28072.582,E2 -28072.582} C_VEL
LIN {X 0,Y 172.206,Z 251.31,A -85,B 0,C 180,E1 -28076.636,E2 -28076.636} C_VEL
LIN {X 0,Y 171.547,Z 248.355,A -85,B 0,C 180,E1 -28082.348,E2 -28082.348} C_VEL
LIN {X 0,Y 171.535,Z 248.511,A -85,B 0,C 180,E1 -28083.56,E2 -28083.56} C_VEL
LIN {X 0,Y 172.415,Z 252.078,A -85,B 0,C 180,E1 -28089.953,E2 -28089.953} C_VEL
LIN {X 0,Y 173.752,Z 255.616,A -85,B 0,C 180,E1 -28093.672,E2 -28093.672} C_VEL
LIN {X 0,Y 174.85,Z 258.64,A -85,B 0,C 180,E1 -28095.959,E2 -28095.959} C_VEL
LIN {X 0,Y 175.302,Z 260.38,A -85,B 0,C 180,E1 -28096.869,E2 -28096.869} C_VEL
LIN {X 0,Y 173.148,Z 275.314,A -85,B 0,C 180,E1 -28097.265,E2 -28097.265} C_VEL
LIN {X 0,Y 169.726,Z 289.496,A -85,B 0,C 180,E1 -28097.751,E2 -28097.751} C_VEL
LIN {X 0,Y 164.867,Z 303.658,A -85,B 0,C 180,E1 -28098.471,E2 -28098.471} C_VEL
LIN {X 0,Y 159.25,Z 316.307,A -85,B 0,C 180,E1 -28099.383,E2 -28099.383} C_VEL
LIN {X 0,Y 152.068,Z 329.223,A -85,B 0,C 180,E1 -28100.629,E2 -28100.629} C_VEL
LIN {X 0,Y 144.199,Z 340.855,A -85,B 0,C 180,E1 -28102.176,E2 -28102.176} C_VEL
LIN {X 0,Y 136.486,Z 350.501,A -85,B 0,C 180,E1 -28103.936,E2 -28103.936} C_VEL
LIN {X 0,Y 127.222,Z 360.425,A -85,B 0,C 180,E1 -28106.453,E2 -28106.453} C_VEL
LIN {X 0,Y 117.294,Z 369.434,A -85,B 0,C 180,E1 -28109.678,E2 -28109.678} C_VEL
LIN {X 0,Y 108.875,Z 375.924,A -85,B 0,C 180,E1 -28112.947,E2 -28112.947} C_VEL
LIN {X 0,Y 100.971,Z 381.326,A -85,B 0,C 180,E1 -28116.826,E2 -28116.826} C_VEL
LIN {X 0,Y 91.25,Z 387.027,A -85,B 0,C 180,E1 -28122.971,E2 -28122.971} C_VEL
LIN {X 0,Y 84.824,Z 390.288,A -85,B 0,C 180,E1 -28128.483,E2 -28128.483} C_VEL
LIN {X 0,Y 77.806,Z 393.368,A -85,B 0,C 180,E1 -28137.182,E2 -28137.182} C_VEL
LIN {X 0,Y 72.689,Z 395.101,A -85,B 0,C 180,E1 -28147.247,E2 -28147.247} C_VEL
LIN {X 0,Y 70.045,Z 395.522,A -85,B 0,C 180,E1 -28158.423,E2 -28158.423} C_VEL
LIN {X 0,Y 69.603,Z 395.24,A -85,B 0,C 180,E1 -28164.204,E2 -28164.204} C_VEL
LIN {X 0,Y 69.639,Z 394.624,A -85,B 0,C 180,E1 -28169.999,E2 -28169.999} C_VEL
LIN {X 0,Y 69.565,Z 393.651,A -85,B 0,C 180,E1 -28175.797,E2 -28175.797} C_VEL
LIN {X 0,Y 70.968,Z 390.649,A -85,B 0,C 180,E1 -28187.282,E2 -28187.282} C_VEL
LIN {X 0,Y 74.731,Z 386.171,A -85,B 0,C 180,E1 -28198.047,E2 -28198.047} C_VEL
LIN {X 0,Y 78.956,Z 381.719,A -85,B 0,C 180,E1 -28205.349,E2 -28205.349} C_VEL
LIN {X 0,Y 85.24,Z 375.271,A -85,B 0,C 180,E1 -28212.859,E2 -28212.859} C_VEL
LIN {X 0,Y 92.776,Z 367.25,A -85,B 0,C 180,E1 -28219.245,E2 -28219.245} C_VEL
LIN {X 0,Y 100.044,Z 358.856,A -85,B 0,C 180,E1 -28223.887,E2 -28223.887} C_VEL
LIN {X 0,Y 107.908,Z 348.744,A -85,B 0,C 180,E1 -28227.851,E2 -28227.851} C_VEL
LIN {X 0,Y 115.251,Z 337.784,A -85,B 0,C 180,E1 -28230.96,E2 -28230.96} C_VEL
LIN {X 0,Y 121.878,Z 326.168,A -85,B 0,C 180,E1 -28233.353,E2 -28233.353} C_VEL
LIN {X 0,Y 127.771,Z 313.877,A -85,B 0,C 180,E1 -28235.171,E2 -28235.171} C_VEL
LIN {X 0,Y 132.681,Z 301.348,A -85,B 0,C 180,E1 -28236.494,E2 -28236.494} C_VEL
LIN {X 0,Y 136.834,Z 287.34,A -85,B 0,C 180,E1 -28237.593,E2 -28237.593} C_VEL
LIN {X 0,Y 139.915,Z 272.514,A -85,B 0,C 180,E1 -28238.346,E2 -28238.346} C_VEL
LIN {X 0,Y 141.589,Z 259.235,A -85,B 0,C 180,E1 -28238.778,E2 -28238.778} C_VEL
LIN {X 0,Y 141.706,Z 255.361,A -85,B 0,C 180,E1 -28239.143,E2 -28239.143} C_VEL
LIN {X 0,Y 140.711,Z 243.402,A -85,B 0,C 180,E1 -28241.654,E2 -28241.654} C_VEL
LIN {X 0,Y 140.851,Z 239.529,A -85,B 0,C 180,E1 -28242.042,E2 -28242.042} C_VEL
LIN {X 0,Y 141.026,Z 236.993,A -85,B 0,C 180,E1 -28242.21,E2 -28242.21} C_VEL
LIN {X 0,Y 138.645,Z 230.902,A -85,B 0,C 180,E1 -28245.974,E2 -28245.974} C_VEL
LIN {X 0,Y 136.449,Z 225.799,A -85,B 0,C 180,E1 -28250.411,E2 -28250.411} C_VEL
LIN {X 0,Y 134.849,Z 221.894,A -85,B 0,C 180,E1 -28255.255,E2 -28255.255} C_VEL
LIN {X 0,Y 133.977,Z 218.591,A -85,B 0,C 180,E1 -28263.007,E2 -28263.007} C_VEL
LIN {X 0,Y 134.759,Z 222.056,A -85,B 0,C 180,E1 -28270.898,E2 -28270.898} C_VEL
LIN {X 0,Y 135.285,Z 223.355,A -85,B 0,C 180,E1 -28272.82,E2 -28272.82} C_VEL
LIN {X 0,Y 136.577,Z 226.238,A -85,B 0,C 180,E1 -28276.3,E2 -28276.3} C_VEL
LIN {X 0,Y 138.232,Z 230.083,A -85,B 0,C 180,E1 -28279.692,E2 -28279.692} C_VEL
LIN {X 0,Y 140.379,Z 235.403,A -85,B 0,C 180,E1 -28283.232,E2 -28283.232} C_VEL
LIN {X 0,Y 141.023,Z 237.12,A -85,B 0,C 180,E1 -28284.18,E2 -28284.18} C_VEL
LIN {X 0,Y 137.595,Z 268.309,A -85,B 0,C 180,E1 -28285.145,E2 -28285.145} C_VEL
LIN {X 0,Y 134.779,Z 282.766,A -85,B 0,C 180,E1 -28285.912,E2 -28285.912} C_VEL
LIN {X 0,Y 131.021,Z 295.987,A -85,B 0,C 180,E1 -28286.905,E2 -28286.905} C_VEL
LIN {X 0,Y 125.747,Z 309.866,A -85,B 0,C 180,E1 -28288.326,E2 -28288.326} C_VEL
LIN {X 0,Y 119.763,Z 322.289,A -85,B 0,C 180,E1 -28290.054,E2 -28290.054} C_VEL
LIN {X 0,Y 112.539,Z 334.785,A -85,B 0,C 180,E1 -28292.536,E2 -28292.536} C_VEL
LIN {X 0,Y 105.542,Z 345.003,A -85,B 0,C 180,E1 -28295.342,E2 -28295.342} C_VEL
LIN {X 0,Y 97.435,Z 355.183,A -85,B 0,C 180,E1 -28299.16,E2 -28299.16} C_VEL
LIN {X 0,Y 89.803,Z 363.609,A -85,B 0,C 180,E1 -28303.623,E2 -28303.623} C_VEL
LIN {X 0,Y 81.774,Z 371.651,A -85,B 0,C 180,E1 -28309.867,E2 -28309.867} C_VEL
LIN {X 0,Y 75.684,Z 377.32,A -85,B 0,C 180,E1 -28316.141,E2 -28316.141} C_VEL
LIN {X 0,Y 69.04,Z 383.289,A -85,B 0,C 180,E1 -28325.973,E2 -28325.973} C_VEL
LIN {X 0,Y 64.645,Z 387.675,A -85,B 0,C 180,E1 -28337.443,E2 -28337.443} C_VEL
LIN {X 0,Y 62.602,Z 390.633,A -85,B 0,C 180,E1 -28350.001,E2 -28350.001} C_VEL
LIN {X 0,Y 62.301,Z 391.61,A -85,B 0,C 180,E1 -28356.478,E2 -28356.478} C_VEL
LIN {X 0,Y 63.435,Z 392.572,A -85,B 0,C 180,E1 -28369.414,E2 -28369.414} C_VEL
LIN {X 0,Y 67.269,Z 392.204,A -85,B 0,C 180,E1 -28381.493,E2 -28381.493} C_VEL
LIN {X 0,Y 73.428,Z 390.492,A -85,B 0,C 180,E1 -28392.067,E2 -28392.067} C_VEL
LIN {X 0,Y 81.562,Z 387.39,A -85,B 0,C 180,E1 -28400.852,E2 -28400.852} C_VEL
LIN {X 0,Y 91.219,Z 382.77,A -85,B 0,C 180,E1 -28407.942,E2 -28407.942} C_VEL
LIN {X 0,Y 101.985,Z 376.466,A -85,B 0,C 180,E1 -28413.62,E2 -28413.62} C_VEL
LIN {X 0,Y 111.948,Z 369.464,A -85,B 0,C 180,E1 -28417.714,E2 -28417.714} C_VEL
LIN {X 0,Y 121.019,Z 362.016,A -85,B 0,C 180,E1 -28420.682,E2 -28420.682} C_VEL
LIN {X 0,Y 130.327,Z 353.097,A -85,B 0,C 180,E1 -28423.174,E2 -28423.174} C_VEL
LIN {X 0,Y 138.259,Z 344.231,A -85,B 0,C 180,E1 -28424.975,E2 -28424.975} C_VEL
LIN {X 0,Y 146.264,Z 333.621,A -85,B 0,C 180,E1 -28426.66,E2 -28426.66} C_VEL
LIN {X 0,Y 153.618,Z 322.042,A -85,B 0,C 180,E1 -28427.934,E2 -28427.934} C_VEL
LIN {X 0,Y 159.354,Z 311.073,A -85,B 0,C 180,E1 -28428.902,E2 -28428.902} C_VEL
LIN {X 0,Y 164.746,Z 298.266,A -85,B 0,C 180,E1 -28429.751,E2 -28429.751} C_VEL
LIN {X 0,Y 169.199,Z 284.177,A -85,B 0,C 180,E1 -28430.473,E2 -28430.473} C_VEL
LIN {X 0,Y 172.292,Z 270.231,A -85,B 0,C 180,E1 -28430.909,E2 -28430.909} C_VEL
LIN {X 0,Y 173.185,Z 264.416,A -85,B 0,C 180,E1 -28431.055,E2 -28431.055} C_VEL
LIN {X 0,Y 171.946,Z 260.594,A -85,B 0,C 180,E1 -28434.355,E2 -28434.355} C_VEL
LIN {X 0,Y 171.145,Z 258.096,A -85,B 0,C 180,E1 -28437.352,E2 -28437.352} C_VEL
LIN {X 0,Y 170.665,Z 255.525,A -85,B 0,C 180,E1 -28442.36,E2 -28442.36} C_VEL
LIN {X 0,Y 170.649,Z 255.718,A -85,B 0,C 180,E1 -28443.578,E2 -28443.578} C_VEL
LIN {X 0,Y 171.38,Z 258.943,A -85,B 0,C 180,E1 -28449.441,E2 -28449.441} C_VEL
LIN {X 0,Y 172.517,Z 262.309,A -85,B 0,C 180,E1 -28452.959,E2 -28452.959} C_VEL
LIN {X 0,Y 173.242,Z 264.443,A -85,B 0,C 180,E1 -28454.709,E2 -28454.709} C_VEL
LIN {X 0,Y 170.618,Z 279.399,A -85,B 0,C 180,E1 -28455.088,E2 -28455.088} C_VEL
LIN {X 0,Y 166.846,Z 293.161,A -85,B 0,C 180,E1 -28455.574,E2 -28455.574} C_VEL
LIN {X 0,Y 161.949,Z 306.316,A -85,B 0,C 180,E1 -28456.238,E2 -28456.238} C_VEL
LIN {X 0,Y 156.226,Z 318.383,A -85,B 0,C 180,E1 -28457.067,E2 -28457.067} C_VEL
LIN {X 0,Y 148.901,Z 330.891,A -85,B 0,C 180,E1 -28458.215,E2 -28458.215} C_VEL
LIN {X 0,Y 140.88,Z 342.207,A -85,B 0,C 180,E1 -28459.676,E2 -28459.676} C_VEL
LIN {X 0,Y 132.202,Z 352.483,A -85,B 0,C 180,E1 -28461.515,E2 -28461.515} C_VEL
LIN {X 0,Y 122.958,Z 361.784,A -85,B 0,C 180,E1 -28463.861,E2 -28463.861} C_VEL
LIN {X 0,Y 112.459,Z 370.666,A -85,B 0,C 180,E1 -28467.058,E2 -28467.058} C_VEL
LIN {X 0,Y 102.358,Z 377.871,A -85,B 0,C 180,E1 -28470.877,E2 -28470.877} C_VEL
LIN {X 0,Y 91.57,Z 384.362,A -85,B 0,C 180,E1 -28476.304,E2 -28476.304} C_VEL
LIN {X 0,Y 84.139,Z 388.166,A -85,B 0,C 180,E1 -28481.257,E2 -28481.257} C_VEL
LIN {X 0,Y 75.547,Z 391.911,A -85,B 0,C 180,E1 -28489.367,E2 -28489.367} C_VEL
LIN {X 0,Y 68.725,Z 394.277,A -85,B 0,C 180,E1 -28499.248,E2 -28499.248} C_VEL
LIN {X 0,Y 64.302,Z 395.32,A -85,B 0,C 180,E1 -28510.858,E2 -28510.858} C_VEL
LIN {X 0,Y 62.535,Z 395.052,A -85,B 0,C 180,E1 -28523.546,E2 -28523.546} C_VEL
LIN {X 0,Y 62.537,Z 394.42,A -85,B 0,C 180,E1 -28529.999,E2 -28529.999} C_VEL
LIN {X 0,Y 62.503,Z 393.43,A -85,B 0,C 180,E1 -28536.455,E2 -28536.455} C_VEL
LIN {X 0,Y 64.173,Z 390.392,A -85,B 0,C 180,E1 -28549.179,E2 -28549.179} C_VEL
LIN {X 0,Y 68.489,Z 385.877,A -85,B 0,C 180,E1 -28560.868,E2 -28560.868} C_VEL
LIN {X 0,Y 73.227,Z 381.387,A -85,B 0,C 180,E1 -28568.596,E2 -28568.596} C_VEL
LIN {X 0,Y 80.133,Z 374.898,A -85,B 0,C 180,E1 -28576.348,E2 -28576.348} C_VEL
LIN {X 0,Y 88.266,Z 366.83,A -85,B 0,C 180,E1 -28582.77,E2 -28582.77} C_VEL
LIN {X 0,Y 96.013,Z 358.386,A -85,B 0,C 180,E1 -28587.327,E2 -28587.327} C_VEL
LIN {X 0,Y 104.289,Z 348.21,A -85,B 0,C 180,E1 -28591.169,E2 -28591.169} C_VEL
LIN {X 0,Y 112.153,Z 336.782,A -85,B 0,C 180,E1 -28594.262,E2 -28594.262} C_VEL
LIN {X 0,Y 118.844,Z 325.413,A -85,B 0,C 180,E1 -28596.434,E2 -28596.434} C_VEL
LIN {X 0,Y 124.945,Z 312.983,A -85,B 0,C 180,E1 -28598.139,E2 -28598.139} C_VEL
LIN {X 0,Y 130.386,Z 299.108,A -85,B 0,C 180,E1 -28599.477,E2 -28599.477} C_VEL
LIN {X 0,Y 134.535,Z 284.872,A -85,B 0,C 180,E1 -28600.475,E2 -28600.475} C_VEL
LIN {X 0,Y 137.448,Z 270.514,A -85,B 0,C 180,E1 -28601.093,E2 -28601.093} C_VEL
LIN {X 0,Y 140.851,Z 239.529,A -85,B 0,C 180,E1 -28602.042,E2 -28602.042} C_VEL
LIN {X 0,Y 140.821,Z 237.135,A -85,B 0,C 180,E1 -28602.409,E2 -28602.409} C_VEL
LIN {X 0,Y 140.228,Z 234.689,A -85,B 0,C 180,E1 -28603.42,E2 -28603.42} C_VEL
LIN {X 0,Y 139.04,Z 232.753,A -85,B 0,C 180,E1 -28605.15,E2 -28605.15} C_VEL
LIN {X 0,Y 137.993,Z 231.995,A -85,B 0,C 180,E1 -28606.676,E2 -28606.676} C_VEL
LIN {X 0,Y 134.776,Z 230.978,A -85,B 0,C 180,E1 -28612.499,E2 -28612.499} C_VEL
LIN {X 0,Y 134.128,Z 229.941,A -85,B 0,C 180,E1 -28614.441,E2 -28614.441} C_VEL
LIN {X 0,Y 133.748,Z 228.672,A -85,B 0,C 180,E1 -28616.103,E2 -28616.103} C_VEL
LIN {X 0,Y 133.092,Z 225.789,A -85,B 0,C 180,E1 -28623.027,E2 -28623.027} C_VEL
LIN {X 0,Y 133.949,Z 229.496,A -85,B 0,C 180,E1 -28631.252,E2 -28631.252} C_VEL
LIN {X 0,Y 135.257,Z 232.901,A -85,B 0,C 180,E1 -28635.395,E2 -28635.395} C_VEL
LIN {X 0,Y 136.923,Z 237.156,A -85,B 0,C 180,E1 -28639.113,E2 -28639.113} C_VEL
LIN {X 0,Y 138.252,Z 240.862,A -85,B 0,C 180,E1 -28641.557,E2 -28641.557} C_VEL
LIN {X 0,Y 135.057,Z 268.672,A -85,B 0,C 180,E1 -28642.366,E2 -28642.366} C_VEL
LIN {X 0,Y 132.159,Z 283.045,A -85,B 0,C 180,E1 -28643.086,E2 -28643.086} C_VEL
LIN {X 0,Y 128.375,Z 295.995,A -85,B 0,C 180,E1 -28643.998,E2 -28643.998} C_VEL
LIN {X 0,Y 123.334,Z 309.028,A -85,B 0,C 180,E1 -28645.23,E2 -28645.23} C_VEL
LIN {X 0,Y 117.163,Z 321.643,A -85,B 0,C 180,E1 -28646.841,E2 -28646.841} C_VEL
LIN {X 0,Y 111.159,Z 331.947,A -85,B 0,C 180,E1 -28648.69,E2 -28648.69} C_VEL
LIN {X 0,Y 104.463,Z 341.716,A -85,B 0,C 180,E1 -28650.933,E2 -28650.933} C_VEL
LIN {X 0,Y 97.32,Z 350.87,A -85,B 0,C 180,E1 -28653.854,E2 -28653.854} C_VEL
LIN {X 0,Y 89.044,Z 360.043,A -85,B 0,C 180,E1 -28657.884,E2 -28657.884} C_VEL
LIN {X 0,Y 81.315,Z 367.689,A -85,B 0,C 180,E1 -28662.724,E2 -28662.724} C_VEL
LIN {X 0,Y 74.228,Z 374.033,A -85,B 0,C 180,E1 -28668.49,E2 -28668.49} C_VEL
LIN {X 0,Y 67.931,Z 379.28,A -85,B 0,C 180,E1 -28675.319,E2 -28675.319} C_VEL
LIN {X 0,Y 61.19,Z 384.822,A -85,B 0,C 180,E1 -28686.298,E2 -28686.298} C_VEL
LIN {X 0,Y 57.76,Z 387.936,A -85,B 0,C 180,E1 -28695.917,E2 -28695.917} C_VEL
LIN {X 0,Y 55.486,Z 390.859,A -85,B 0,C 180,E1 -28710.001,E2 -28710.001} C_VEL
LIN {X 0,Y 55.196,Z 391.818,A -85,B 0,C 180,E1 -28717.316,E2 -28717.316} C_VEL
LIN {X 0,Y 56.694,Z 392.747,A -85,B 0,C 180,E1 -28731.833,E2 -28731.833} C_VEL
LIN {X 0,Y 61.247,Z 392.342,A -85,B 0,C 180,E1 -28745.013,E2 -28745.013} C_VEL
LIN {X 0,Y 68.221,Z 390.596,A -85,B 0,C 180,E1 -28756.149,E2 -28756.149} C_VEL
LIN {X 0,Y 77.201,Z 387.454,A -85,B 0,C 180,E1 -28765.018,E2 -28765.018} C_VEL
LIN {X 0,Y 87.602,Z 382.78,A -85,B 0,C 180,E1 -28771.945,E2 -28771.945} C_VEL
LIN {X 0,Y 98.982,Z 376.433,A -85,B 0,C 180,E1 -28777.375,E2 -28777.375} C_VEL
LIN {X 0,Y 109.858,Z 369.066,A -85,B 0,C 180,E1 -28781.344,E2 -28781.344} C_VEL
LIN {X 0,Y 120.412,Z 360.522,A -85,B 0,C 180,E1 -28784.376,E2 -28784.376} C_VEL
LIN {X 0,Y 130.063,Z 351.269,A -85,B 0,C 180,E1 -28786.566,E2 -28786.566} C_VEL
LIN {X 0,Y 138.575,Z 341.55,A -85,B 0,C 180,E1 -28788.295,E2 -28788.295} C_VEL
LIN {X 0,Y 146.428,Z 330.905,A -85,B 0,C 180,E1 -28789.714,E2 -28789.714} C_VEL
LIN {X 0,Y 153.941,Z 318.686,A -85,B 0,C 180,E1 -28790.849,E2 -28790.849} C_VEL
LIN {X 0,Y 159.812,Z 306.899,A -85,B 0,C 180,E1 -28791.681,E2 -28791.681} C_VEL
LIN {X 0,Y 165.227,Z 292.889,A -85,B 0,C 180,E1 -28792.465,E2 -28792.465} C_VEL
LIN {X 0,Y 169.123,Z 279.121,A -85,B 0,C 180,E1 -28793.025,E2 -28793.025} C_VEL
LIN {X 0,Y 171.144,Z 269.117,A -85,B 0,C 180,E1 -28793.323,E2 -28793.323} C_VEL
LIN {X 0,Y 170.509,Z 266.694,A -85,B 0,C 180,E1 -28795.715,E2 -28795.715} C_VEL
LIN {X 0,Y 170.084,Z 264.967,A -85,B 0,C 180,E1 -28797.854,E2 -28797.854} C_VEL
LIN {X 0,Y 169.771,Z 262.691,A -85,B 0,C 180,E1 -28802.372,E2 -28802.372} C_VEL
LIN {X 0,Y 169.748,Z 262.922,A -85,B 0,C 180,E1 -28803.597,E2 -28803.597} C_VEL
LIN {X 0,Y 170.306,Z 265.935,A -85,B 0,C 180,E1 -28809.052,E2 -28809.052} C_VEL
LIN {X 0,Y 171.162,Z 268.892,A -85,B 0,C 180,E1 -28812.205,E2 -28812.205} C_VEL
LIN {X 0,Y 171.24,Z 269.186,A -85,B 0,C 180,E1 -28812.456,E2 -28812.456} C_VEL
LIN {X 0,Y 168.206,Z 283.63,A -85,B 0,C 180,E1 -28812.844,E2 -28812.844} C_VEL
LIN {X 0,Y 164.104,Z 296.954,A -85,B 0,C 180,E1 -28813.34,E2 -28813.34} C_VEL
LIN {X 0,Y 159.296,Z 308.864,A -85,B 0,C 180,E1 -28813.921,E2 -28813.921} C_VEL
LIN {X 0,Y 153.465,Z 320.435,A -85,B 0,C 180,E1 -28814.663,E2 -28814.663} C_VEL
LIN {X 0,Y 146.019,Z 332.481,A -85,B 0,C 180,E1 -28815.715,E2 -28815.715} C_VEL
LIN {X 0,Y 137.832,Z 343.464,A -85,B 0,C 180,E1 -28817.047,E2 -28817.047} C_VEL
LIN {X 0,Y 128.177,Z 354.297,A -85,B 0,C 180,E1 -28818.944,E2 -28818.944} C_VEL
LIN {X 0,Y 118.688,Z 363.26,A -85,B 0,C 180,E1 -28821.151,E2 -28821.151} C_VEL
LIN {X 0,Y 107.88,Z 371.852,A -85,B 0,C 180,E1 -28824.209,E2 -28824.209} C_VEL
LIN {X 0,Y 98.888,Z 377.898,A -85,B 0,C 180,E1 -28827.329,E2 -28827.329} C_VEL
LIN {X 0,Y 87.546,Z 384.349,A -85,B 0,C 180,E1 -28832.549,E2 -28832.549} C_VEL
LIN {X 0,Y 77.122,Z 389.184,A -85,B 0,C 180,E1 -28839.231,E2 -28839.231} C_VEL
LIN {X 0,Y 70.282,Z 391.823,A -85,B 0,C 180,E1 -28845.574,E2 -28845.574} C_VEL
LIN {X 0,Y 62.71,Z 394.155,A -85,B 0,C 180,E1 -28855.919,E2 -28855.919} C_VEL
LIN {X 0,Y 57.596,Z 395.164,A -85,B 0,C 180,E1 -28868.526,E2 -28868.526} C_VEL
LIN {X 0,Y 55.469,Z 394.864,A -85,B 0,C 180,E1 -28882.72,E2 -28882.72} C_VEL
LIN {X 0,Y 55.454,Z 394.216,A -85,B 0,C 180,E1 -28889.999,E2 -28889.999} C_VEL
LIN {X 0,Y 55.438,Z 393.209,A -85,B 0,C 180,E1 -28897.282,E2 -28897.282} C_VEL
LIN {X 0,Y 57.478,Z 390.136,A -85,B 0,C 180,E1 -28911.518,E2 -28911.518} C_VEL
LIN {X 0,Y 62.453,Z 385.583,A -85,B 0,C 180,E1 -28924.239,E2 -28924.239} C_VEL
LIN {X 0,Y 67.768,Z 381.055,A -85,B 0,C 180,E1 -28932.383,E2 -28932.383} C_VEL
LIN {X 0,Y 75.363,Z 374.524,A -85,B 0,C 180,E1 -28940.295,E2 -28940.295} C_VEL
LIN {X 0,Y 84.132,Z 366.41,A -85,B 0,C 180,E1 -28946.651,E2 -28946.651} C_VEL
LIN {X 0,Y 92.352,Z 357.912,A -85,B 0,C 180,E1 -28951.061,E2 -28951.061} C_VEL
LIN {X 0,Y 101.047,Z 347.657,A -85,B 0,C 180,E1 -28954.71,E2 -28954.71} C_VEL
LIN {X 0,Y 109.242,Z 336.124,A -85,B 0,C 180,E1 -28957.637,E2 -28957.637} C_VEL
LIN {X 0,Y 116.179,Z 324.649,A -85,B 0,C 180,E1 -28959.657,E2 -28959.657} C_VEL
LIN {X 0,Y 122.469,Z 312.073,A -85,B 0,C 180,E1 -28961.236,E2 -28961.236} C_VEL
LIN {X 0,Y 128.07,Z 297.994,A -85,B 0,C 180,E1 -28962.452,E2 -28962.452} C_VEL
LIN {X 0,Y 132.215,Z 283.784,A -85,B 0,C 180,E1 -28963.383,E2 -28963.383} C_VEL
LIN {X 0,Y 135.115,Z 269.423,A -85,B 0,C 180,E1 -28963.92,E2 -28963.92} C_VEL
LIN {X 0,Y 138.292,Z 241.108,A -85,B 0,C 180,E1 -28964.73,E2 -28964.73} C_VEL
LIN {X 0,Y 136.931,Z 237.061,A -85,B 0,C 180,E1 -28967.269,E2 -28967.269} C_VEL
LIN {X 0,Y 134.981,Z 232.005,A -85,B 0,C 180,E1 -28971.769,E2 -28971.769} C_VEL
LIN {X 0,Y 134.128,Z 229.941,A -85,B 0,C 180,E1 -28974.441,E2 -28974.441} C_VEL
LIN {X 0,Y 133.689,Z 229.209,A -85,B 0,C 180,E1 -28976.076,E2 -28976.076} C_VEL
LIN {X 0,Y 133.056,Z 229.493,A -85,B 0,C 180,E1 -28978.602,E2 -28978.602} C_VEL
LIN {X 0,Y 132.321,Z 232.074,A -85,B 0,C 180,E1 -28982.815,E2 -28982.815} C_VEL
LIN {X 0,Y 132.214,Z 234.435,A -85,B 0,C 180,E1 -28986.246,E2 -28986.246} C_VEL
LIN {X 0,Y 132.395,Z 235.198,A -85,B 0,C 180,E1 -28987.997,E2 -28987.997} C_VEL
LIN {X 0,Y 132.922,Z 236.512,A -85,B 0,C 180,E1 -28990.761,E2 -28990.761} C_VEL
LIN {X 0,Y 134.027,Z 239.718,A -85,B 0,C 180,E1 -28994.634,E2 -28994.634} C_VEL
LIN {X 0,Y 135.382,Z 243.589,A -85,B 0,C 180,E1 -28998.006,E2 -28998.006} C_VEL
LIN {X 0,Y 135.772,Z 244.806,A -85,B 0,C 180,E1 -28998.855,E2 -28998.855} C_VEL
LIN {X 0,Y 132.817,Z 269.237,A -85,B 0,C 180,E1 -28999.503,E2 -28999.503} C_VEL
LIN {X 0,Y 129.836,Z 283.459,A -85,B 0,C 180,E1 -29000.16,E2 -29000.16} C_VEL
LIN {X 0,Y 125.669,Z 297.128,A -85,B 0,C 180,E1 -29001.056,E2 -29001.056} C_VEL
LIN {X 0,Y 120.495,Z 309.949,A -85,B 0,C 180,E1 -29002.193,E2 -29002.193} C_VEL
LIN {X 0,Y 114.152,Z 322.416,A -85,B 0,C 180,E1 -29003.681,E2 -29003.681} C_VEL
LIN {X 0,Y 107.948,Z 332.613,A -85,B 0,C 180,E1 -29005.401,E2 -29005.401} C_VEL
LIN {X 0,Y 101.01,Z 342.297,A -85,B 0,C 180,E1 -29007.49,E2 -29007.49} C_VEL
LIN {X 0,Y 93.566,Z 351.381,A -85,B 0,C 180,E1 -29010.256,E2 -29010.256} C_VEL
LIN {X 0,Y 84.879,Z 360.497,A -85,B 0,C 180,E1 -29014.107,E2 -29014.107} C_VEL
LIN {X 0,Y 76.685,Z 368.094,A -85,B 0,C 180,E1 -29018.832,E2 -29018.832} C_VEL
LIN {X 0,Y 69.095,Z 374.412,A -85,B 0,C 180,E1 -29024.603,E2 -29024.603} C_VEL
LIN {X 0,Y 62.24,Z 379.616,A -85,B 0,C 180,E1 -29031.609,E2 -29031.609} C_VEL
LIN {X 0,Y 54.782,Z 385.118,A -85,B 0,C 180,E1 -29043.321,E2 -29043.321} C_VEL
LIN {X 0,Y 50.925,Z 388.194,A -85,B 0,C 180,E1 -29053.979,E2 -29053.979} C_VEL
LIN {X 0,Y 48.359,Z 391.083,A -85,B 0,C 180,E1 -29070.001,E2 -29070.001} C_VEL
LIN {X 0,Y 48.658,Z 392.639,A -85,B 0,C 180,E1 -29086.792,E2 -29086.792} C_VEL
LIN {X 0,Y 52.424,Z 392.867,A -85,B 0,C 180,E1 -29102.43,E2 -29102.43} C_VEL
LIN {X 0,Y 59.187,Z 391.761,A -85,B 0,C 180,E1 -29115.437,E2 -29115.437} C_VEL
LIN {X 0,Y 68.155,Z 389.29,A -85,B 0,C 180,E1 -29125.585,E2 -29125.585} C_VEL
LIN {X 0,Y 78.737,Z 385.349,A -85,B 0,C 180,E1 -29133.202,E2 -29133.202} C_VEL
LIN {X 0,Y 90.361,Z 379.814,A -85,B 0,C 180,E1 -29138.961,E2 -29138.961} C_VEL
LIN {X 0,Y 101.078,Z 373.531,A -85,B 0,C 180,E1 -29142.951,E2 -29142.951} C_VEL
LIN {X 0,Y 112.182,Z 365.677,A -85,B 0,C 180,E1 -29146.182,E2 -29146.182} C_VEL
LIN {X 0,Y 121.963,Z 357.448,A -85,B 0,C 180,E1 -29148.412,E2 -29148.412} C_VEL
LIN {X 0,Y 131.915,Z 347.505,A -85,B 0,C 180,E1 -29150.274,E2 -29150.274} C_VEL
LIN {X 0,Y 141.024,Z 336.513,A -85,B 0,C 180,E1 -29151.857,E2 -29151.857} C_VEL
LIN {X 0,Y 148.719,Z 325.373,A -85,B 0,C 180,E1 -29152.933,E2 -29152.933} C_VEL
LIN {X 0,Y 155.515,Z 313.379,A -85,B 0,C 180,E1 -29153.838,E2 -29153.838} C_VEL
LIN {X 0,Y 161.49,Z 300.127,A -85,B 0,C 180,E1 -29154.572,E2 -29154.572} C_VEL
LIN {X 0,Y 166.311,Z 285.819,A -85,B 0,C 180,E1 -29155.206,E2 -29155.206} C_VEL
LIN {X 0,Y 169.203,Z 274.047,A -85,B 0,C 180,E1 -29155.567,E2 -29155.567} C_VEL
LIN {X 0,Y 168.815,Z 271.871,A -85,B 0,C 180,E1 -29158.211,E2 -29158.211} C_VEL
LIN {X 0,Y 168.673,Z 269.807,A -85,B 0,C 180,E1 -29162.388,E2 -29162.388} C_VEL
LIN {X 0,Y 168.622,Z 270.208,A -85,B 0,C 180,E1 -29163.827,E2 -29163.827} C_VEL
LIN {X 0,Y 168.968,Z 272.725,A -85,B 0,C 180,E1 -29168.521,E2 -29168.521} C_VEL
LIN {X 0,Y 169.272,Z 274.175,A -85,B 0,C 180,E1 -29170.225,E2 -29170.225} C_VEL
LIN {X 0,Y 165.876,Z 287.984,A -85,B 0,C 180,E1 -29170.577,E2 -29170.577} C_VEL
LIN {X 0,Y 160.86,Z 302.315,A -85,B 0,C 180,E1 -29171.08,E2 -29171.08} C_VEL
LIN {X 0,Y 155.196,Z 314.66,A -85,B 0,C 180,E1 -29171.682,E2 -29171.682} C_VEL
LIN {X 0,Y 147.63,Z 327.784,A -85,B 0,C 180,E1 -29172.599,E2 -29172.599} C_VEL
LIN {X 0,Y 139.261,Z 339.58,A -85,B 0,C 180,E1 -29173.715,E2 -29173.715} C_VEL
LIN {X 0,Y 130.968,Z 349.358,A -85,B 0,C 180,E1 -29175,E2 -29175} C_VEL
LIN {X 0,Y 120.732,Z 359.52,A -85,B 0,C 180,E1 -29176.921,E2 -29176.921} C_VEL
LIN {X 0,Y 109.918,Z 368.49,A -85,B 0,C 180,E1 -29179.421,E2 -29179.421} C_VEL
LIN {X 0,Y 98.9,Z 376.069,A -85,B 0,C 180,E1 -29182.51,E2 -29182.51} C_VEL
LIN {X 0,Y 89.802,Z 381.343,A -85,B 0,C 180,E1 -29185.841,E2 -29185.841} C_VEL
LIN {X 0,Y 78.241,Z 386.925,A -85,B 0,C 180,E1 -29191.422,E2 -29191.422} C_VEL
LIN {X 0,Y 69.579,Z 390.301,A -85,B 0,C 180,E1 -29197.303,E2 -29197.303} C_VEL
LIN {X 0,Y 60.886,Z 393.052,A -85,B 0,C 180,E1 -29206.164,E2 -29206.164} C_VEL
LIN {X 0,Y 53.561,Z 394.684,A -85,B 0,C 180,E1 -29218.34,E2 -29218.34} C_VEL
LIN {X 0,Y 49.285,Z 395.007,A -85,B 0,C 180,E1 -29233.428,E2 -29233.428} C_VEL
LIN {X 0,Y 48.353,Z 394.012,A -85,B 0,C 180,E1 -29249.999,E2 -29249.999} C_VEL
LIN {X 0,Y 48.382,Z 392.987,A -85,B 0,C 180,E1 -29258.351,E2 -29258.351} C_VEL
LIN {X 0,Y 50.907,Z 389.879,A -85,B 0,C 180,E1 -29274.465,E2 -29274.465} C_VEL
LIN {X 0,Y 56.684,Z 385.28,A -85,B 0,C 180,E1 -29288.309,E2 -29288.309} C_VEL
LIN {X 0,Y 62.641,Z 380.719,A -85,B 0,C 180,E1 -29296.823,E2 -29296.823} C_VEL
LIN {X 0,Y 71.004,Z 374.146,A -85,B 0,C 180,E1 -29304.743,E2 -29304.743} C_VEL
LIN {X 0,Y 80.415,Z 365.983,A -85,B 0,C 180,E1 -29310.922,E2 -29310.922} C_VEL
LIN {X 0,Y 89.105,Z 357.431,A -85,B 0,C 180,E1 -29315.098,E2 -29315.098} C_VEL
LIN {X 0,Y 98.215,Z 347.085,A -85,B 0,C 180,E1 -29318.47,E2 -29318.47} C_VEL
LIN {X 0,Y 106.71,Z 335.459,A -85,B 0,C 180,E1 -29321.215,E2 -29321.215} C_VEL
LIN {X 0,Y 113.899,Z 323.884,A -85,B 0,C 180,E1 -29323.019,E2 -29323.019} C_VEL
LIN {X 0,Y 120.361,Z 311.161,A -85,B 0,C 180,E1 -29324.459,E2 -29324.459} C_VEL
LIN {X 0,Y 125.69,Z 298.012,A -85,B 0,C 180,E1 -29325.471,E2 -29325.471} C_VEL
LIN {X 0,Y 130.057,Z 283.444,A -85,B 0,C 180,E1 -29326.335,E2 -29326.335} C_VEL
LIN {X 0,Y 132.864,Z 269.921,A -85,B 0,C 180,E1 -29326.784,E2 -29326.784} C_VEL
LIN {X 0,Y 135.798,Z 244.772,A -85,B 0,C 180,E1 -29327.488,E2 -29327.488} C_VEL
LIN {X 0,Y 134.096,Z 239.851,A -85,B 0,C 180,E1 -29331.56,E2 -29331.56} C_VEL
LIN {X 0,Y 133.341,Z 237.714,A -85,B 0,C 180,E1 -29333.949,E2 -29333.949} C_VEL
LIN {X 0,Y 132.673,Z 235.479,A -85,B 0,C 180,E1 -29336.964,E2 -29336.964} C_VEL
LIN {X 0,Y 132.21,Z 232.963,A -85,B 0,C 180,E1 -29343.048,E2 -29343.048} C_VEL
LIN {X 0,Y 132.395,Z 235.198,A -85,B 0,C 180,E1 -29347.997,E2 -29347.997} C_VEL
LIN {X 0,Y 132.595,Z 236.472,A -85,B 0,C 180,E1 -29349.584,E2 -29349.584} C_VEL
LIN {X 0,Y 132.706,Z 238.787,A -85,B 0,C 180,E1 -29350.974,E2 -29350.974} C_VEL
LIN {X 0,Y 133.042,Z 246.499,A -85,B 0,C 180,E1 -29354.344,E2 -29354.344} C_VEL
LIN {X 0,Y 133.3,Z 248.091,A -85,B 0,C 180,E1 -29355.304,E2 -29355.304} C_VEL
LIN {X 0,Y 133.541,Z 248.902,A -85,B 0,C 180,E1 -29355.974,E2 -29355.974} C_VEL
LIN {X 0,Y 131.072,Z 268.942,A -85,B 0,C 180,E1 -29356.515,E2 -29356.515} C_VEL
LIN {X 0,Y 127.989,Z 283.424,A -85,B 0,C 180,E1 -29357.12,E2 -29357.12} C_VEL
LIN {X 0,Y 123.72,Z 297.137,A -85,B 0,C 180,E1 -29357.92,E2 -29357.92} C_VEL
LIN {X 0,Y 118.008,Z 310.87,A -85,B 0,C 180,E1 -29359.016,E2 -29359.016} C_VEL
LIN {X 0,Y 111.498,Z 323.192,A -85,B 0,C 180,E1 -29360.348,E2 -29360.348} C_VEL
LIN {X 0,Y 104.313,Z 334.447,A -85,B 0,C 180,E1 -29362.122,E2 -29362.122} C_VEL
LIN {X 0,Y 96.42,Z 344.811,A -85,B 0,C 180,E1 -29364.342,E2 -29364.342} C_VEL
LIN {X 0,Y 87.155,Z 355.127,A -85,B 0,C 180,E1 -29367.502,E2 -29367.502} C_VEL
LIN {X 0,Y 78.174,Z 363.643,A -85,B 0,C 180,E1 -29371.344,E2 -29371.344} C_VEL
LIN {X 0,Y 68.313,Z 371.789,A -85,B 0,C 180,E1 -29377.127,E2 -29377.127} C_VEL
LIN {X 0,Y 59.251,Z 378.348,A -85,B 0,C 180,E1 -29384.63,E2 -29384.63} C_VEL
LIN {X 0,Y 50.379,Z 384.18,A -85,B 0,C 180,E1 -29396.084,E2 -29396.084} C_VEL
LIN {X 0,Y 44.153,Z 388.453,A -85,B 0,C 180,E1 -29411.438,E2 -29411.438} C_VEL
LIN {X 0,Y 41.217,Z 391.308,A -85,B 0,C 180,E1 -29430.002,E2 -29430.002} C_VEL
LIN {X 0,Y 41.037,Z 392.234,A -85,B 0,C 180,E1 -29439.863,E2 -29439.863} C_VEL
LIN {X 0,Y 43.663,Z 393.094,A -85,B 0,C 180,E1 -29458.875,E2 -29458.875} C_VEL
LIN {X 0,Y 50.119,Z 392.621,A -85,B 0,C 180,E1 -29474.519,E2 -29474.519} C_VEL
LIN {X 0,Y 59.125,Z 390.803,A -85,B 0,C 180,E1 -29486.314,E2 -29486.314} C_VEL
LIN {X 0,Y 69.915,Z 387.564,A -85,B 0,C 180,E1 -29494.785,E2 -29494.785} C_VEL
LIN {X 0,Y 81.804,Z 382.799,A -85,B 0,C 180,E1 -29500.917,E2 -29500.917} C_VEL
LIN {X 0,Y 94.367,Z 376.367,A -85,B 0,C 180,E1 -29505.509,E2 -29505.509} C_VEL
LIN {X 0,Y 104.564,Z 369.973,A -85,B 0,C 180,E1 -29508.367,E2 -29508.367} C_VEL
LIN {X 0,Y 115.678,Z 361.622,A -85,B 0,C 180,E1 -29510.849,E2 -29510.849} C_VEL
LIN {X 0,Y 125.796,Z 352.526,A -85,B 0,C 180,E1 -29512.598,E2 -29512.598} C_VEL
LIN {X 0,Y 135.669,Z 341.852,A -85,B 0,C 180,E1 -29514.124,E2 -29514.124} C_VEL
LIN {X 0,Y 143.699,Z 331.394,A -85,B 0,C 180,E1 -29515.204,E2 -29515.204} C_VEL
LIN {X 0,Y 151.457,Z 319.22,A -85,B 0,C 180,E1 -29516.081,E2 -29516.081} C_VEL
LIN {X 0,Y 157.509,Z 307.476,A -85,B 0,C 180,E1 -29516.73,E2 -29516.73} C_VEL
LIN {X 0,Y 162.833,Z 294.366,A -85,B 0,C 180,E1 -29517.321,E2 -29517.321} C_VEL
LIN {X 0,Y 167.004,Z 280.432,A -85,B 0,C 180,E1 -29517.786,E2 -29517.786} C_VEL
LIN {X 0,Y 167.275,Z 279.274,A -85,B 0,C 180,E1 -29517.817,E2 -29517.817} C_VEL
LIN {X 0,Y 167.137,Z 277.629,A -85,B 0,C 180,E1 -29520.903,E2 -29520.903} C_VEL
LIN {X 0,Y 167.241,Z 276.845,A -85,B 0,C 180,E1 -29523.011,E2 -29523.011} C_VEL
LIN {X 0,Y 167.33,Z 279.372,A -85,B 0,C 180,E1 -29527.904,E2 -29527.904} C_VEL
LIN {X 0,Y 163.345,Z 293.217,A -85,B 0,C 180,E1 -29528.275,E2 -29528.275} C_VEL
LIN {X 0,Y 157.975,Z 306.861,A -85,B 0,C 180,E1 -29528.742,E2 -29528.742} C_VEL
LIN {X 0,Y 151.368,Z 319.872,A -85,B 0,C 180,E1 -29529.375,E2 -29529.375} C_VEL
LIN {X 0,Y 143.69,Z 331.969,A -85,B 0,C 180,E1 -29530.155,E2 -29530.155} C_VEL
LIN {X 0,Y 134.363,Z 343.957,A -85,B 0,C 180,E1 -29531.262,E2 -29531.262} C_VEL
LIN {X 0,Y 124.293,Z 354.655,A -85,B 0,C 180,E1 -29532.738,E2 -29532.738} C_VEL
LIN {X 0,Y 114.338,Z 363.502,A -85,B 0,C 180,E1 -29534.509,E2 -29534.509} C_VEL
LIN {X 0,Y 102.876,Z 371.995,A -85,B 0,C 180,E1 -29536.977,E2 -29536.977} C_VEL
LIN {X 0,Y 93.215,Z 377.952,A -85,B 0,C 180,E1 -29539.533,E2 -29539.533} C_VEL
LIN {X 0,Y 80.763,Z 384.322,A -85,B 0,C 180,E1 -29543.975,E2 -29543.975} C_VEL
LIN {X 0,Y 71.841,Z 388.011,A -85,B 0,C 180,E1 -29548.303,E2 -29548.303} C_VEL
LIN {X 0,Y 60.89,Z 391.648,A -85,B 0,C 180,E1 -29556.102,E2 -29556.102} C_VEL
LIN {X 0,Y 51.498,Z 393.911,A -85,B 0,C 180,E1 -29566.97,E2 -29566.97} C_VEL
LIN {X 0,Y 44.625,Z 394.854,A -85,B 0,C 180,E1 -29581.803,E2 -29581.803} C_VEL
LIN {X 0,Y 41.391,Z 394.487,A -85,B 0,C 180,E1 -29600.223,E2 -29600.223} C_VEL
LIN {X 0,Y 41.248,Z 393.807,A -85,B 0,C 180,E1 -29609.998,E2 -29609.998} C_VEL
LIN {X 0,Y 41.362,Z 392.765,A -85,B 0,C 180,E1 -29619.781,E2 -29619.781} C_VEL
LIN {X 0,Y 44.496,Z 389.62,A -85,B 0,C 180,E1 -29638.282,E2 -29638.282} C_VEL
LIN {X 0,Y 51.262,Z 384.969,A -85,B 0,C 180,E1 -29653.273,E2 -29653.273} C_VEL
LIN {X 0,Y 60.046,Z 378.89,A -85,B 0,C 180,E1 -29664.183,E2 -29664.183} C_VEL
LIN {X 0,Y 69.936,Z 371.574,A -85,B 0,C 180,E1 -29671.557,E2 -29671.557} C_VEL
LIN {X 0,Y 80.174,Z 362.815,A -85,B 0,C 180,E1 -29676.986,E2 -29676.986} C_VEL
LIN {X 0,Y 89.476,Z 353.665,A -85,B 0,C 180,E1 -29680.482,E2 -29680.482} C_VEL
LIN {X 0,Y 98.396,Z 343.312,A -85,B 0,C 180,E1 -29683.227,E2 -29683.227} C_VEL
LIN {X 0,Y 106.257,Z 332.43,A -85,B 0,C 180,E1 -29685.309,E2 -29685.309} C_VEL
LIN {X 0,Y 113.673,Z 320.229,A -85,B 0,C 180,E1 -29686.845,E2 -29686.845} C_VEL
LIN {X 0,Y 119.486,Z 308.47,A -85,B 0,C 180,E1 -29687.918,E2 -29687.918} C_VEL
LIN {X 0,Y 124.814,Z 294.792,A -85,B 0,C 180,E1 -29688.801,E2 -29688.801} C_VEL
LIN {X 0,Y 128.857,Z 280.609,A -85,B 0,C 180,E1 -29689.449,E2 -29689.449} C_VEL
LIN {X 0,Y 131.632,Z 265.735,A -85,B 0,C 180,E1 -29689.868,E2 -29689.868} C_VEL
LIN {X 0,Y 133.567,Z 248.927,A -85,B 0,C 180,E1 -29690.345,E2 -29690.345} C_VEL
LIN {X 0,Y 132.385,Z 244.941,A -85,B 0,C 180,E1 -29694.097,E2 -29694.097} C_VEL
LIN {X 0,Y 131.652,Z 242.323,A -85,B 0,C 180,E1 -29697.706,E2 -29697.706} C_VEL
LIN {X 0,Y 131.324,Z 240.167,A -85,B 0,C 180,E1 -29703.068,E2 -29703.068} C_VEL
LIN {X 0,Y 131.854,Z 243.292,A -85,B 0,C 180,E1 -29709.976,E2 -29709.976} C_VEL
LIN {X 0,Y 132.753,Z 246.318,A -85,B 0,C 180,E1 -29713.637,E2 -29713.637} C_VEL
LIN {X 0,Y 133.3,Z 248.091,A -85,B 0,C 180,E1 -29715.304,E2 -29715.304} C_VEL
LIN {X 0,Y 133.442,Z 249.969,A -85,B 0,C 180,E1 -29716.026,E2 -29716.026} C_VEL
LIN {X 0,Y 133.255,Z 253.331,A -85,B 0,C 180,E1 -29716.429,E2 -29716.429} C_VEL
LIN {X 0,Y 132.589,Z 258.05,A -85,B 0,C 180,E1 -29716.284,E2 -29716.284} C_VEL
LIN {X 0,Y 131.845,Z 261.748,A -85,B 0,C 180,E1 -29715.84,E2 -29715.84} C_VEL
LIN {X 0,Y 129.237,Z 272.431,A -85,B 0,C 180,E1 -29714.104,E2 -29714.104} C_VEL
LIN {X 0,Y 128.127,Z 276.829,A -85,B 0,C 180,E1 -29713.776,E2 -29713.776} C_VEL
LIN {X 0,Y 127.583,Z 279.06,A -85,B 0,C 180,E1 -29713.795,E2 -29713.795} C_VEL
LIN {X 0,Y 124.027,Z 291.719,A -85,B 0,C 180,E1 -29714.367,E2 -29714.367} C_VEL
LIN {X 0,Y 119.239,Z 304.488,A -85,B 0,C 180,E1 -29715.174,E2 -29715.174} C_VEL
LIN {X 0,Y 112.564,Z 318.218,A -85,B 0,C 180,E1 -29716.274,E2 -29716.274} C_VEL
LIN {X 0,Y 105.115,Z 330.448,A -85,B 0,C 180,E1 -29717.685,E2 -29717.685} C_VEL
LIN {X 0,Y 96.944,Z 341.519,A -85,B 0,C 180,E1 -29719.537,E2 -29719.537} C_VEL
LIN {X 0,Y 88.918,Z 350.764,A -85,B 0,C 180,E1 -29721.767,E2 -29721.767} C_VEL
LIN {X 0,Y 79.391,Z 360.054,A -85,B 0,C 180,E1 -29724.858,E2 -29724.858} C_VEL
LIN {X 0,Y 70.192,Z 367.767,A -85,B 0,C 180,E1 -29728.827,E2 -29728.827} C_VEL
LIN {X 0,Y 60.007,Z 375.153,A -85,B 0,C 180,E1 -29734.934,E2 -29734.934} C_VEL
LIN {X 0,Y 51.885,Z 380.288,A -85,B 0,C 180,E1 -29741.844,E2 -29741.844} C_VEL
LIN {X 0,Y 42.599,Z 385.708,A -85,B 0,C 180,E1 -29754.732,E2 -29754.732} C_VEL
LIN {X 0,Y 37.492,Z 388.712,A -85,B 0,C 180,E1 -29767.983,E2 -29767.983} C_VEL
LIN {X 0,Y 35.244,Z 390.293,A -85,B 0,C 180,E1 -29778.499,E2 -29778.499} C_VEL
LIN {X 0,Y 34.081,Z 391.532,A -85,B 0,C 180,E1 -29790.002,E2 -29790.002} C_VEL
LIN {X 0,Y 35.167,Z 393.02,A -85,B 0,C 180,E1 -29813.561,E2 -29813.561} C_VEL
LIN {X 0,Y 40.98,Z 393.181,A -85,B 0,C 180,E1 -29833.316,E2 -29833.316} C_VEL
LIN {X 0,Y 50.092,Z 392.004,A -85,B 0,C 180,E1 -29847.334,E2 -29847.334} C_VEL
LIN {X 0,Y 61.146,Z 389.44,A -85,B 0,C 180,E1 -29856.856,E2 -29856.856} C_VEL
LIN {X 0,Y 73.364,Z 385.408,A -85,B 0,C 180,E1 -29863.331,E2 -29863.331} C_VEL
LIN {X 0,Y 86.229,Z 379.791,A -85,B 0,C 180,E1 -29867.976,E2 -29867.976} C_VEL
LIN {X 0,Y 97.817,Z 373.42,A -85,B 0,C 180,E1 -29871.088,E2 -29871.088} C_VEL
LIN {X 0,Y 109.633,Z 365.468,A -85,B 0,C 180,E1 -29873.531,E2 -29873.531} C_VEL
LIN {X 0,Y 119.902,Z 357.128,A -85,B 0,C 180,E1 -29875.172,E2 -29875.172} C_VEL
LIN {X 0,Y 129.934,Z 347.39,A -85,B 0,C 180,E1 -29876.496,E2 -29876.496} C_VEL
LIN {X 0,Y 138.925,Z 336.888,A -85,B 0,C 180,E1 -29877.61,E2 -29877.61} C_VEL
LIN {X 0,Y 146.769,Z 325.878,A -85,B 0,C 180,E1 -29878.374,E2 -29878.374} C_VEL
LIN {X 0,Y 153.759,Z 313.924,A -85,B 0,C 180,E1 -29879.05,E2 -29879.05} C_VEL
LIN {X 0,Y 159.821,Z 300.938,A -85,B 0,C 180,E1 -29879.588,E2 -29879.588} C_VEL
LIN {X 0,Y 164.695,Z 287.112,A -85,B 0,C 180,E1 -29880.067,E2 -29880.067} C_VEL
LIN {X 0,Y 165.316,Z 284.922,A -85,B 0,C 180,E1 -29880.152,E2 -29880.152} C_VEL
LIN {X 0,Y 165.466,Z 283.847,A -85,B 0,C 180,E1 -29882.434,E2 -29882.434} C_VEL
LIN {X 0,Y 165.369,Z 284.338,A -85,B 0,C 180,E1 -29883.96,E2 -29883.96} C_VEL
LIN {X 0,Y 165.322,Z 285.1,A -85,B 0,C 180,E1 -29885.555,E2 -29885.555} C_VEL
LIN {X 0,Y 160.505,Z 299.398,A -85,B 0,C 180,E1 -29885.949,E2 -29885.949} C_VEL
LIN {X 0,Y 154.693,Z 312.355,A -85,B 0,C 180,E1 -29886.368,E2 -29886.368} C_VEL
LIN {X 0,Y 147.786,Z 324.586,A -85,B 0,C 180,E1 -29886.916,E2 -29886.916} C_VEL
LIN {X 0,Y 140.033,Z 335.808,A -85,B 0,C 180,E1 -29887.596,E2 -29887.596} C_VEL
LIN {X 0,Y 131.449,Z 346.148,A -85,B 0,C 180,E1 -29888.461,E2 -29888.461} C_VEL
LIN {X 0,Y 121.222,Z 356.453,A -85,B 0,C 180,E1 -29889.733,E2 -29889.733} C_VEL
LIN {X 0,Y 111.08,Z 364.974,A -85,B 0,C 180,E1 -29891.278,E2 -29891.278} C_VEL
LIN {X 0,Y 99.358,Z 373.143,A -85,B 0,C 180,E1 -29893.442,E2 -29893.442} C_VEL
LIN {X 0,Y 87.804,Z 379.74,A -85,B 0,C 180,E1 -29896.154,E2 -29896.154} C_VEL
LIN {X 0,Y 74.973,Z 385.614,A -85,B 0,C 180,E1 -29900.378,E2 -29900.378} C_VEL
LIN {X 0,Y 62.714,Z 389.936,A -85,B 0,C 180,E1 -29906.294,E2 -29906.294} C_VEL
LIN {X 0,Y 51.53,Z 392.842,A -85,B 0,C 180,E1 -29915.081,E2 -29915.081} C_VEL
LIN {X 0,Y 42.073,Z 394.406,A -85,B 0,C 180,E1 -29928.071,E2 -29928.071} C_VEL
LIN {X 0,Y 35.85,Z 394.663,A -85,B 0,C 180,E1 -29946.914,E2 -29946.914} C_VEL
LIN {X 0,Y 34.133,Z 393.601,A -85,B 0,C 180,E1 -29969.998,E2 -29969.998} C_VEL
LIN {X 0,Y 34.361,Z 392.542,A -85,B 0,C 180,E1 -29981.8,E2 -29981.8} C_VEL
LIN {X 0,Y 38.334,Z 389.36,A -85,B 0,C 180,E1 -30003.365,E2 -30003.365} C_VEL
LIN {X 0,Y 46.301,Z 384.654,A -85,B 0,C 180,E1 -30019.369,E2 -30019.369} C_VEL
LIN {X 0,Y 55.442,Z 379.004,A -85,B 0,C 180,E1 -30029.533,E2 -30029.533} C_VEL
LIN {X 0,Y 65.315,Z 372.301,A -85,B 0,C 180,E1 -30036.149,E2 -30036.149} C_VEL
LIN {X 0,Y 76.071,Z 363.732,A -85,B 0,C 180,E1 -30041.254,E2 -30041.254} C_VEL
LIN {X 0,Y 85.724,Z 354.799,A -85,B 0,C 180,E1 -30044.429,E2 -30044.429} C_VEL
LIN {X 0,Y 94.862,Z 344.792,A -85,B 0,C 180,E1 -30046.858,E2 -30046.858} C_VEL
LIN {X 0,Y 102.989,Z 334.132,A -85,B 0,C 180,E1 -30048.796,E2 -30048.796} C_VEL
LIN {X 0,Y 110.572,Z 322.35,A -85,B 0,C 180,E1 -30050.121,E2 -30050.121} C_VEL
LIN {X 0,Y 117.348,Z 309.342,A -85,B 0,C 180,E1 -30051.182,E2 -30051.182} C_VEL
LIN {X 0,Y 122.878,Z 295.774,A -85,B 0,C 180,E1 -30051.948,E2 -30051.948} C_VEL
LIN {X 0,Y 127.054,Z 281.872,A -85,B 0,C 180,E1 -30052.507,E2 -30052.507} C_VEL
LIN {X 0,Y 129.923,Z 267.585,A -85,B 0,C 180,E1 -30052.869,E2 -30052.869} C_VEL
LIN {X 0,Y 131.677,Z 253.435,A -85,B 0,C 180,E1 -30053.187,E2 -30053.187} C_VEL
LIN {X 0,Y 131.027,Z 250.949,A -85,B 0,C 180,E1 -30055.964,E2 -30055.964} C_VEL
LIN {X 0,Y 130.657,Z 249.149,A -85,B 0,C 180,E1 -30058.459,E2 -30058.459} C_VEL
LIN {X 0,Y 130.436,Z 247.385,A -85,B 0,C 180,E1 -30063.089,E2 -30063.089} C_VEL
LIN {X 0,Y 130.795,Z 250.02,A -85,B 0,C 180,E1 -30069.082,E2 -30069.082} C_VEL
LIN {X 0,Y 131.507,Z 252.868,A -85,B 0,C 180,E1 -30072.572,E2 -30072.572} C_VEL
LIN {X 0,Y 131.642,Z 253.353,A -85,B 0,C 180,E1 -30073.076,E2 -30073.076} C_VEL
LIN {X 0,Y 129.445,Z 269.974,A -85,B 0,C 180,E1 -30073.488,E2 -30073.488} C_VEL
LIN {X 0,Y 127.583,Z 279.06,A -85,B 0,C 180,E1 -30073.795,E2 -30073.795} C_VEL
LIN {X 0,Y 126.043,Z 284.774,A -85,B 0,C 180,E1 -30073.724,E2 -30073.724} C_VEL
LIN {X 0,Y 122.762,Z 293.957,A -85,B 0,C 180,E1 -30072.857,E2 -30072.857} C_VEL
LIN {X 0,Y 118.877,Z 302.903,A -85,B 0,C 180,E1 -30072.011,E2 -30072.011} C_VEL
LIN {X 0,Y 116.351,Z 308.244,A -85,B 0,C 180,E1 -30072.021,E2 -30072.021} C_VEL
LIN {X 0,Y 109.953,Z 320.482,A -85,B 0,C 180,E1 -30072.906,E2 -30072.906} C_VEL
LIN {X 0,Y 102.361,Z 332.283,A -85,B 0,C 180,E1 -30074.119,E2 -30074.119} C_VEL
LIN {X 0,Y 93.143,Z 344.041,A -85,B 0,C 180,E1 -30075.842,E2 -30075.842} C_VEL
LIN {X 0,Y 84.887,Z 352.915,A -85,B 0,C 180,E1 -30077.805,E2 -30077.805} C_VEL
LIN {X 0,Y 75.074,Z 361.856,A -85,B 0,C 180,E1 -30080.589,E2 -30080.589} C_VEL
LIN {X 0,Y 65.503,Z 369.3,A -85,B 0,C 180,E1 -30084.221,E2 -30084.221} C_VEL
LIN {X 0,Y 56.248,Z 375.513,A -85,B 0,C 180,E1 -30089.001,E2 -30089.001} C_VEL
LIN {X 0,Y 47.463,Z 380.623,A -85,B 0,C 180,E1 -30095.474,E2 -30095.474} C_VEL
LIN {X 0,Y 37.045,Z 385.994,A -85,B 0,C 180,E1 -30108.397,E2 -30108.397} C_VEL
LIN {X 0,Y 31.048,Z 388.97,A -85,B 0,C 180,E1 -30123.085,E2 -30123.085} C_VEL
LIN {X 0,Y 26.961,Z 391.756,A -85,B 0,C 180,E1 -30150.002,E2 -30150.002} C_VEL
LIN {X 0,Y 28.728,Z 393.211,A -85,B 0,C 180,E1 -30179.296,E2 -30179.296} C_VEL
LIN {X 0,Y 36.07,Z 393.338,A -85,B 0,C 180,E1 -30201.206,E2 -30201.206} C_VEL
LIN {X 0,Y 46.588,Z 392.119,A -85,B 0,C 180,E1 -30214.843,E2 -30214.843} C_VEL
LIN {X 0,Y 58.681,Z 389.508,A -85,B 0,C 180,E1 -30223.366,E2 -30223.366} C_VEL
LIN {X 0,Y 71.623,Z 385.438,A -85,B 0,C 180,E1 -30228.889,E2 -30228.889} C_VEL
LIN {X 0,Y 85.017,Z 379.78,A -85,B 0,C 180,E1 -30232.749,E2 -30232.749} C_VEL
LIN {X 0,Y 96.96,Z 373.365,A -85,B 0,C 180,E1 -30235.316,E2 -30235.316} C_VEL
LIN {X 0,Y 109.057,Z 365.364,A -85,B 0,C 180,E1 -30237.293,E2 -30237.293} C_VEL
LIN {X 0,Y 119.512,Z 356.968,A -85,B 0,C 180,E1 -30238.615,E2 -30238.615} C_VEL
LIN {X 0,Y 129.331,Z 347.535,A -85,B 0,C 180,E1 -30239.641,E2 -30239.641} C_VEL
LIN {X 0,Y 138.811,Z 336.583,A -85,B 0,C 180,E1 -30240.585,E2 -30240.585} C_VEL
LIN {X 0,Y 146.741,Z 325.475,A -85,B 0,C 180,E1 -30241.18,E2 -30241.18} C_VEL
LIN {X 0,Y 153.807,Z 313.378,A -85,B 0,C 180,E1 -30241.717,E2 -30241.717} C_VEL
LIN {X 0,Y 159.929,Z 300.13,A -85,B 0,C 180,E1 -30242.152,E2 -30242.152} C_VEL
LIN {X 0,Y 163.373,Z 290.714,A -85,B 0,C 180,E1 -30242.465,E2 -30242.465} C_VEL
LIN {X 0,Y 163.387,Z 290.679,A -85,B 0,C 180,E1 -30242.883,E2 -30242.883} C_VEL
LIN {X 0,Y 162.78,Z 292.509,A -85,B 0,C 180,E1 -30243.279,E2 -30243.279} C_VEL
LIN {X 0,Y 157.205,Z 306.489,A -85,B 0,C 180,E1 -30243.574,E2 -30243.574} C_VEL
LIN {X 0,Y 150.589,Z 319.301,A -85,B 0,C 180,E1 -30243.99,E2 -30243.99} C_VEL
LIN {X 0,Y 142.75,Z 331.457,A -85,B 0,C 180,E1 -30244.461,E2 -30244.461} C_VEL
LIN {X 0,Y 134.065,Z 342.503,A -85,B 0,C 180,E1 -30245.106,E2 -30245.106} C_VEL
LIN {X 0,Y 123.675,Z 353.39,A -85,B 0,C 180,E1 -30246.031,E2 -30246.031} C_VEL
LIN {X 0,Y 112.428,Z 363.116,A -85,B 0,C 180,E1 -30247.328,E2 -30247.328} C_VEL
LIN {X 0,Y 101.366,Z 371.022,A -85,B 0,C 180,E1 -30248.883,E2 -30248.883} C_VEL
LIN {X 0,Y 89.463,Z 378.006,A -85,B 0,C 180,E1 -30250.894,E2 -30250.894} C_VEL
LIN {X 0,Y 76.094,Z 384.295,A -85,B 0,C 180,E1 -30254.12,E2 -30254.12} C_VEL
LIN {X 0,Y 66.28,Z 387.908,A -85,B 0,C 180,E1 -30257.383,E2 -30257.383} C_VEL
LIN {X 0,Y 53.709,Z 391.473,A -85,B 0,C 180,E1 -30263.654,E2 -30263.654} C_VEL
LIN {X 0,Y 42.203,Z 393.668,A -85,B 0,C 180,E1 -30273.626,E2 -30273.626} C_VEL
LIN {X 0,Y 32.743,Z 394.543,A -85,B 0,C 180,E1 -30289.912,E2 -30289.912} C_VEL
LIN {X 0,Y 27.469,Z 394.11,A -85,B 0,C 180,E1 -30315.173,E2 -30315.173} C_VEL
LIN {X 0,Y 27.029,Z 393.396,A -85,B 0,C 180,E1 -30329.998,E2 -30329.998} C_VEL
LIN {X 0,Y 27.413,Z 392.319,A -85,B 0,C 180,E1 -30344.853,E2 -30344.853} C_VEL
LIN {X 0,Y 32.59,Z 389.095,A -85,B 0,C 180,E1 -30370.309,E2 -30370.309} C_VEL
LIN {X 0,Y 41.978,Z 384.338,A -85,B 0,C 180,E1 -30386.833,E2 -30386.833} C_VEL
LIN {X 0,Y 53.4,Z 377.917,A -85,B 0,C 180,E1 -30397.11,E2 -30397.11} C_VEL
LIN {X 0,Y 64.351,Z 370.771,A -85,B 0,C 180,E1 -30402.863,E2 -30402.863} C_VEL
LIN {X 0,Y 74.084,Z 363.281,A -85,B 0,C 180,E1 -30406.496,E2 -30406.496} C_VEL
LIN {X 0,Y 84.085,Z 354.29,A -85,B 0,C 180,E1 -30409.134,E2 -30409.134} C_VEL
LIN {X 0,Y 93.703,Z 343.963,A -85,B 0,C 180,E1 -30411.197,E2 -30411.197} C_VEL
LIN {X 0,Y 101.846,Z 333.475,A -85,B 0,C 180,E1 -30412.724,E2 -30412.724} C_VEL
LIN {X 0,Y 109.574,Z 321.584,A -85,B 0,C 180,E1 -30413.799,E2 -30413.799} C_VEL
LIN {X 0,Y 116.469,Z 308.433,A -85,B 0,C 180,E1 -30414.644,E2 -30414.644} C_VEL
LIN {X 0,Y 121.731,Z 295.583,A -85,B 0,C 180,E1 -30415.224,E2 -30415.224} C_VEL
LIN {X 0,Y 125.896,Z 281.972,A -85,B 0,C 180,E1 -30415.669,E2 -30415.669} C_VEL
LIN {X 0,Y 128.718,Z 268.465,A -85,B 0,C 180,E1 -30415.956,E2 -30415.956} C_VEL
LIN {X 0,Y 130.078,Z 258.126,A -85,B 0,C 180,E1 -30416.174,E2 -30416.174} C_VEL
LIN {X 0,Y 129.681,Z 256.001,A -85,B 0,C 180,E1 -30419.224,E2 -30419.224} C_VEL
LIN {X 0,Y 129.548,Z 254.607,A -85,B 0,C 180,E1 -30423.11,E2 -30423.11} C_VEL
LIN {X 0,Y 129.789,Z 256.893,A -85,B 0,C 180,E1 -30428.368,E2 -30428.368} C_VEL
LIN {X 0,Y 130.044,Z 258.152,A -85,B 0,C 180,E1 -30430.09,E2 -30430.09} C_VEL
LIN {X 0,Y 127.668,Z 273.822,A -85,B 0,C 180,E1 -30430.487,E2 -30430.487} C_VEL
LIN {X 0,Y 124.011,Z 288.285,A -85,B 0,C 180,E1 -30430.958,E2 -30430.958} C_VEL
LIN {X 0,Y 119.277,Z 301.556,A -85,B 0,C 180,E1 -30431.603,E2 -30431.603} C_VEL
LIN {X 0,Y 116.351,Z 308.244,A -85,B 0,C 180,E1 -30432.021,E2 -30432.021} C_VEL
LIN {X 0,Y 113.654,Z 313.59,A -85,B 0,C 180,E1 -30432.059,E2 -30432.059} C_VEL
LIN {X 0,Y 108.572,Z 321.973,A -85,B 0,C 180,E1 -30431.261,E2 -30431.261} C_VEL
LIN {X 0,Y 103.079,Z 329.999,A -85,B 0,C 180,E1 -30430.403,E2 -30430.403} C_VEL
LIN {X 0,Y 99.603,Z 334.687,A -85,B 0,C 180,E1 -30430.429,E2 -30430.429} C_VEL
LIN {X 0,Y 91.468,Z 344.623,A -85,B 0,C 180,E1 -30431.582,E2 -30431.582} C_VEL
LIN {X 0,Y 81.309,Z 355.044,A -85,B 0,C 180,E1 -30433.498,E2 -30433.498} C_VEL
LIN {X 0,Y 71.207,Z 363.657,A -85,B 0,C 180,E1 -30435.786,E2 -30435.786} C_VEL
LIN {X 0,Y 59.659,Z 371.914,A -85,B 0,C 180,E1 -30439.541,E2 -30439.541} C_VEL
LIN {X 0,Y 49.992,Z 377.667,A -85,B 0,C 180,E1 -30443.971,E2 -30443.971} C_VEL
LIN {X 0,Y 37.718,Z 383.825,A -85,B 0,C 180,E1 -30453.022,E2 -30453.022} C_VEL
LIN {X 0,Y 29.491,Z 387.333,A -85,B 0,C 180,E1 -30464.366,E2 -30464.366} C_VEL
LIN {X 0,Y 24.925,Z 389.23,A -85,B 0,C 180,E1 -30475.675,E2 -30475.675} C_VEL
LIN {X 0,Y 21.513,Z 390.775,A -85,B 0,C 180,E1 -30490.936,E2 -30490.936} C_VEL
LIN {X 0,Y 19.811,Z 391.982,A -85,B 0,C 180,E1 -30510.003,E2 -30510.003} C_VEL
LIN {X 0,Y 22.724,Z 393.403,A -85,B 0,C 180,E1 -30548.213,E2 -30548.213} C_VEL
LIN {X 0,Y 32.049,Z 393.492,A -85,B 0,C 180,E1 -30571.307,E2 -30571.307} C_VEL
LIN {X 0,Y 44.006,Z 392.228,A -85,B 0,C 180,E1 -30583.388,E2 -30583.388} C_VEL
LIN {X 0,Y 57.034,Z 389.576,A -85,B 0,C 180,E1 -30590.337,E2 -30590.337} C_VEL
LIN {X 0,Y 70.589,Z 385.467,A -85,B 0,C 180,E1 -30594.648,E2 -30594.648} C_VEL
LIN {X 0,Y 84.41,Z 379.769,A -85,B 0,C 180,E1 -30597.617,E2 -30597.617} C_VEL
LIN {X 0,Y 96.638,Z 373.309,A -85,B 0,C 180,E1 -30599.597,E2 -30599.597} C_VEL
LIN {X 0,Y 108.954,Z 365.26,A -85,B 0,C 180,E1 -30601.086,E2 -30601.086} C_VEL
LIN {X 0,Y 119.554,Z 356.808,A -85,B 0,C 180,E1 -30602.062,E2 -30602.062} C_VEL
LIN {X 0,Y 124.752,Z 352.056,A -85,B 0,C 180,E1 -30602.429,E2 -30602.429} C_VEL
LIN {X 0,Y 123.132,Z 353.569,A -85,B 0,C 180,E1 -30602.744,E2 -30602.744} C_VEL
LIN {X 0,Y 112.672,Z 362.515,A -85,B 0,C 180,E1 -30603.611,E2 -30603.611} C_VEL
LIN {X 0,Y 100.513,Z 371.094,A -85,B 0,C 180,E1 -30604.874,E2 -30604.874} C_VEL
LIN {X 0,Y 88.395,Z 378.033,A -85,B 0,C 180,E1 -30606.359,E2 -30606.359} C_VEL
LIN {X 0,Y 74.678,Z 384.281,A -85,B 0,C 180,E1 -30608.822,E2 -30608.822} C_VEL
LIN {X 0,Y 64.511,Z 387.856,A -85,B 0,C 180,E1 -30611.332,E2 -30611.332} C_VEL
LIN {X 0,Y 51.26,Z 391.386,A -85,B 0,C 180,E1 -30616.309,E2 -30616.309} C_VEL
LIN {X 0,Y 38.712,Z 393.547,A -85,B 0,C 180,E1 -30624.802,E2 -30624.802} C_VEL
LIN {X 0,Y 27.656,Z 394.387,A -85,B 0,C 180,E1 -30640.322,E2 -30640.322} C_VEL
LIN {X 0,Y 20.661,Z 393.922,A -85,B 0,C 180,E1 -30670.11,E2 -30670.11} C_VEL
LIN {X 0,Y 19.936,Z 393.192,A -85,B 0,C 180,E1 -30689.997,E2 -30689.997} C_VEL
LIN {X 0,Y 20.609,Z 392.096,A -85,B 0,C 180,E1 -30709.935,E2 -30709.935} C_VEL
LIN {X 0,Y 27.524,Z 388.824,A -85,B 0,C 180,E1 -30739.993,E2 -30739.993} C_VEL
LIN {X 0,Y 38.522,Z 384.022,A -85,B 0,C 180,E1 -30755.807,E2 -30755.807} C_VEL
LIN {X 0,Y 51.049,Z 377.562,A -85,B 0,C 180,E1 -30764.509,E2 -30764.509} C_VEL
LIN {X 0,Y 62.611,Z 370.369,A -85,B 0,C 180,E1 -30769.161,E2 -30769.161} C_VEL
LIN {X 0,Y 72.747,Z 362.831,A -85,B 0,C 180,E1 -30771.982,E2 -30771.982} C_VEL
LIN {X 0,Y 83.033,Z 353.781,A -85,B 0,C 180,E1 -30773.995,E2 -30773.995} C_VEL
LIN {X 0,Y 91.662,Z 344.773,A -85,B 0,C 180,E1 -30775.371,E2 -30775.371} C_VEL
LIN {X 0,Y 100.32,Z 333.997,A -85,B 0,C 180,E1 -30776.644,E2 -30776.644} C_VEL
LIN {X 0,Y 108.162,Z 322.254,A -85,B 0,C 180,E1 -30777.443,E2 -30777.443} C_VEL
LIN {X 0,Y 115.147,Z 309.303,A -85,B 0,C 180,E1 -30778.079,E2 -30778.079} C_VEL
LIN {X 0,Y 120.965,Z 295.457,A -85,B 0,C 180,E1 -30778.547,E2 -30778.547} C_VEL
LIN {X 0,Y 125.25,Z 281.56,A -85,B 0,C 180,E1 -30778.903,E2 -30778.903} C_VEL
LIN {X 0,Y 128.079,Z 268.054,A -85,B 0,C 180,E1 -30779.115,E2 -30779.115} C_VEL
LIN {X 0,Y 128.767,Z 263.22,A -85,B 0,C 180,E1 -30779.243,E2 -30779.243} C_VEL
LIN {X 0,Y 128.667,Z 261.773,A -85,B 0,C 180,E1 -30783.132,E2 -30783.132} C_VEL
LIN {X 0,Y 128.731,Z 263.364,A -85,B 0,C 180,E1 -30787.089,E2 -30787.089} C_VEL
LIN {X 0,Y 126.018,Z 278.111,A -85,B 0,C 180,E1 -30787.389,E2 -30787.389} C_VEL
LIN {X 0,Y 122.166,Z 291.677,A -85,B 0,C 180,E1 -30787.813,E2 -30787.813} C_VEL
LIN {X 0,Y 117.202,Z 304.547,A -85,B 0,C 180,E1 -30788.345,E2 -30788.345} C_VEL
LIN {X 0,Y 111.169,Z 316.756,A -85,B 0,C 180,E1 -30788.963,E2 -30788.963} C_VEL
LIN {X 0,Y 103.431,Z 329.329,A -85,B 0,C 180,E1 -30789.855,E2 -30789.855} C_VEL
LIN {X 0,Y 99.603,Z 334.687,A -85,B 0,C 180,E1 -30790.429,E2 -30790.429} C_VEL
LIN {X 0,Y 95.938,Z 339.353,A -85,B 0,C 180,E1 -30790.471,E2 -30790.471} C_VEL
LIN {X 0,Y 89.341,Z 346.653,A -85,B 0,C 180,E1 -30789.539,E2 -30789.539} C_VEL
LIN {X 0,Y 82.291,Z 353.471,A -85,B 0,C 180,E1 -30788.619,E2 -30788.619} C_VEL
LIN {X 0,Y 77.882,Z 357.374,A -85,B 0,C 180,E1 -30788.842,E2 -30788.842} C_VEL
LIN {X 0,Y 66.189,Z 366.603,A -85,B 0,C 180,E1 -30790.839,E2 -30790.839} C_VEL
LIN {X 0,Y 54.285,Z 374.306,A -85,B 0,C 180,E1 -30793.843,E2 -30793.843} C_VEL
LIN {X 0,Y 44.222,Z 379.691,A -85,B 0,C 180,E1 -30797.535,E2 -30797.535} C_VEL
LIN {X 0,Y 31.178,Z 385.364,A -85,B 0,C 180,E1 -30805.627,E2 -30805.627} C_VEL
LIN {X 0,Y 19.488,Z 389.488,A -85,B 0,C 180,E1 -30823.846,E2 -30823.846} C_VEL
LIN {X 0,Y 14.976,Z 391.017,A -85,B 0,C 180,E1 -30842.017,E2 -30842.017} C_VEL
LIN {X 0,Y 12.677,Z 392.206,A -85,B 0,C 180,E1 -30870.005,E2 -30870.005} C_VEL
LIN {X 0,Y 17.638,Z 393.593,A -85,B 0,C 180,E1 -30922.841,E2 -30922.841} C_VEL
LIN {X 0,Y 29.279,Z 393.639,A -85,B 0,C 180,E1 -30943.774,E2 -30943.774} C_VEL
LIN {X 0,Y 42.505,Z 392.332,A -85,B 0,C 180,E1 -30952.794,E2 -30952.794} C_VEL
LIN {X 0,Y 56.273,Z 389.644,A -85,B 0,C 180,E1 -30957.63,E2 -30957.63} C_VEL
LIN {X 0,Y 70.284,Z 385.497,A -85,B 0,C 180,E1 -30960.51,E2 -30960.51} C_VEL
LIN {X 0,Y 77.339,Z 382.837,A -85,B 0,C 180,E1 -30961.607,E2 -30961.607} C_VEL
LIN {X 0,Y 77.408,Z 382.84,A -85,B 0,C 180,E1 -30962.899,E2 -30962.899} C_VEL
LIN {X 0,Y 63.495,Z 387.805,A -85,B 0,C 180,E1 -30965.006,E2 -30965.006} C_VEL
LIN {X 0,Y 49.725,Z 391.298,A -85,B 0,C 180,E1 -30968.36,E2 -30968.36} C_VEL
LIN {X 0,Y 36.298,Z 393.425,A -85,B 0,C 180,E1 -30974.508,E2 -30974.508} C_VEL
LIN {X 0,Y 23.665,Z 394.232,A -85,B 0,C 180,E1 -30987.002,E2 -30987.002} C_VEL
LIN {X 0,Y 14.179,Z 393.733,A -85,B 0,C 180,E1 -31020.282,E2 -31020.282} C_VEL
LIN {X 0,Y 12.831,Z 392.986,A -85,B 0,C 180,E1 -31049.995,E2 -31049.995} C_VEL
LIN {X 0,Y 14.131,Z 391.87,A -85,B 0,C 180,E1 -31079.819,E2 -31079.819} C_VEL
LIN {X 0,Y 23.572,Z 388.547,A -85,B 0,C 180,E1 -31113.429,E2 -31113.429} C_VEL
LIN {X 0,Y 36.179,Z 383.706,A -85,B 0,C 180,E1 -31126.226,E2 -31126.226} C_VEL
LIN {X 0,Y 46.895,Z 378.663,A -85,B 0,C 180,E1 -31131.606,E2 -31131.606} C_VEL
LIN {X 0,Y 58.212,Z 372.227,A -85,B 0,C 180,E1 -31134.878,E2 -31134.878} C_VEL
LIN {X 0,Y 68.61,Z 365.096,A -85,B 0,C 180,E1 -31137.096,E2 -31137.096} C_VEL
LIN {X 0,Y 79.09,Z 356.54,A -85,B 0,C 180,E1 -31138.511,E2 -31138.511} C_VEL
LIN {X 0,Y 89.607,Z 346.168,A -85,B 0,C 180,E1 -31139.652,E2 -31139.652} C_VEL
LIN {X 0,Y 98.396,Z 335.698,A -85,B 0,C 180,E1 -31140.623,E2 -31140.623} C_VEL
LIN {X 0,Y 106.318,Z 324.357,A -85,B 0,C 180,E1 -31141.133,E2 -31141.133} C_VEL
LIN {X 0,Y 113.367,Z 311.948,A -85,B 0,C 180,E1 -31141.55,E2 -31141.55} C_VEL
LIN {X 0,Y 119.537,Z 298.1,A -85,B 0,C 180,E1 -31141.855,E2 -31141.855} C_VEL
LIN {X 0,Y 124.095,Z 284.443,A -85,B 0,C 180,E1 -31142.144,E2 -31142.144} C_VEL
LIN {X 0,Y 127.408,Z 270.091,A -85,B 0,C 180,E1 -31142.261,E2 -31142.261} C_VEL
LIN {X 0,Y 127.597,Z 269.101,A -85,B 0,C 180,E1 -31142.307,E2 -31142.307} C_VEL
LIN {X 0,Y 127.593,Z 269.04,A -85,B 0,C 180,E1 -31143.385,E2 -31143.385} C_VEL
LIN {X 0,Y 127.554,Z 269.289,A -85,B 0,C 180,E1 -31143.99,E2 -31143.99} C_VEL
LIN {X 0,Y 124.359,Z 283.479,A -85,B 0,C 180,E1 -31144.307,E2 -31144.307} C_VEL
LIN {X 0,Y 119.869,Z 297.175,A -85,B 0,C 180,E1 -31144.649,E2 -31144.649} C_VEL
LIN {X 0,Y 113.776,Z 311.039,A -85,B 0,C 180,E1 -31145.101,E2 -31145.101} C_VEL
LIN {X 0,Y 106.81,Z 323.451,A -85,B 0,C 180,E1 -31145.619,E2 -31145.619} C_VEL
LIN {X 0,Y 99.863,Z 333.613,A -85,B 0,C 180,E1 -31146.251,E2 -31146.251} C_VEL
LIN {X 0,Y 92.046,Z 343.265,A -85,B 0,C 180,E1 -31146.984,E2 -31146.984} C_VEL
LIN {X 0,Y 83.414,Z 352.318,A -85,B 0,C 180,E1 -31148.121,E2 -31148.121} C_VEL
LIN {X 0,Y 77.882,Z 357.374,A -85,B 0,C 180,E1 -31148.842,E2 -31148.842} C_VEL
LIN {X 0,Y 73.327,Z 361.17,A -85,B 0,C 180,E1 -31149.095,E2 -31149.095} C_VEL
LIN {X 0,Y 65.42,Z 366.959,A -85,B 0,C 180,E1 -31147.948,E2 -31147.948} C_VEL
LIN {X 0,Y 57.192,Z 372.295,A -85,B 0,C 180,E1 -31146.462,E2 -31146.462} C_VEL
LIN {X 0,Y 52.069,Z 375.215,A -85,B 0,C 180,E1 -31146.565,E2 -31146.565} C_VEL
LIN {X 0,Y 39.164,Z 381.623,A -85,B 0,C 180,E1 -31149.264,E2 -31149.264} C_VEL
LIN {X 0,Y 25.431,Z 386.827,A -85,B 0,C 180,E1 -31154.72,E2 -31154.72} C_VEL
LIN {X 0,Y 15.447,Z 389.747,A -85,B 0,C 180,E1 -31164.511,E2 -31164.511} C_VEL
LIN {X 0,Y 9.327,Z 391.258,A -85,B 0,C 180,E1 -31181.113,E2 -31181.113} C_VEL
LIN {X 0,Y 5.529,Z 392.431,A -85,B 0,C 180,E1 -31230.012,E2 -31230.012} C_VEL
LIN {X 0,Y 14.475,Z 393.778,A -85,B 0,C 180,E1 -31306.198,E2 -31306.198} C_VEL
LIN {X 0,Y 28.13,Z 393.781,A -85,B 0,C 180,E1 -31318.005,E2 -31318.005} C_VEL
LIN {X 0,Y 35.143,Z 393.277,A -85,B 0,C 180,E1 -31320.675,E2 -31320.675} C_VEL
LIN {X 0,Y 35.194,Z 393.303,A -85,B 0,C 180,E1 -31323.152,E2 -31323.152} C_VEL
LIN {X 0,Y 21.39,Z 394.076,A -85,B 0,C 180,E1 -31329.679,E2 -31329.679} C_VEL
LIN {X 0,Y 8.749,Z 393.543,A -85,B 0,C 180,E1 -31356.545,E2 -31356.545} C_VEL
LIN {X 0,Y 5.718,Z 392.776,A -85,B 0,C 180,E1 -31409.988,E2 -31409.988} C_VEL
LIN {X 0,Y 8.694,Z 391.636,A -85,B 0,C 180,E1 -31463.926,E2 -31463.926} C_VEL
LIN {X 0,Y 21.354,Z 388.271,A -85,B 0,C 180,E1 -31490.862,E2 -31490.862} C_VEL
LIN {X 0,Y 35.169,Z 383.391,A -85,B 0,C 180,E1 -31497.642,E2 -31497.642} C_VEL
LIN {X 0,Y 45.895,Z 378.566,A -85,B 0,C 180,E1 -31500.299,E2 -31500.299} C_VEL
LIN {X 0,Y 58.014,Z 371.826,A -85,B 0,C 180,E1 -31501.957,E2 -31501.957} C_VEL
LIN {X 0,Y 68.62,Z 364.659,A -85,B 0,C 180,E1 -31503.075,E2 -31503.075} C_VEL
LIN {X 0,Y 70.389,Z 363.294,A -85,B 0,C 180,E1 -31503.209,E2 -31503.209} C_VEL
LIN {X 0,Y 70.469,Z 363.216,A -85,B 0,C 180,E1 -31504.211,E2 -31504.211} C_VEL
LIN {X 0,Y 60.001,Z 370.508,A -85,B 0,C 180,E1 -31505.379,E2 -31505.379} C_VEL
LIN {X 0,Y 52.069,Z 375.215,A -85,B 0,C 180,E1 -31506.565,E2 -31506.565} C_VEL
LIN {X 0,Y 51.032,Z 376.975,A -85,B 0,C 180,E1 -31506.746,E2 -31506.746} C_VEL
LIN {X 0,Y 51.032,Z 600,A -85,B 0,C 180,E1 -31506.746,E2 -31506.746} C_VEL
LIN {X 0,Y 51.032,Z 600,A -85,B 0,C 180,E1 -31506.746,E2 -31506.746}

QRS_NEXT_CUT()

QRS_NEXT()
QRS_HOME()

END
